KUKA KRL program: MyProgram_001().src

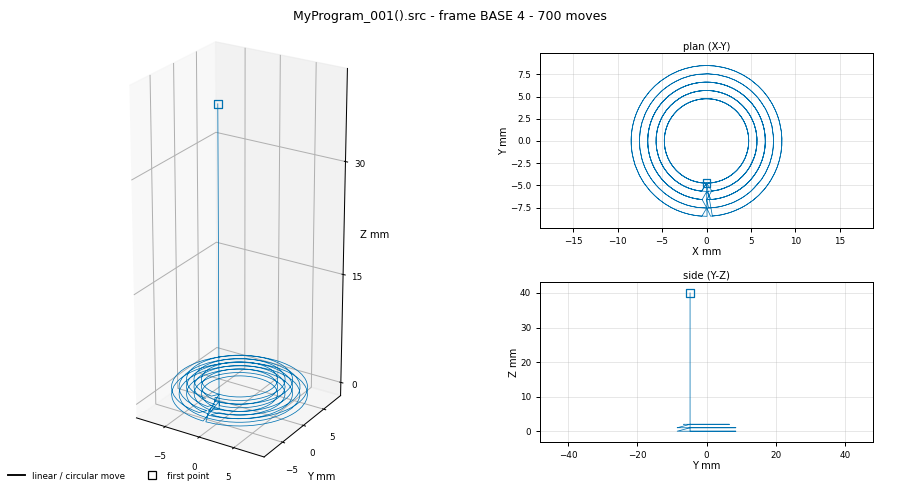
[picture p0: tool path of MyProgram_001().src in frame BASE 4, 700 of 700 moves have a stored position in this frame; points joined in program order, loops and branches not executed]
&ACCESS RVP
&REL 1
&PARAM TEMPLATE = C:\KRC\Roboter\Template\vorgabe
&PARAM EDITMASK = *
DEF MyProgram_001()
; ---- Setting reference (Base) ----
$BASE = BASE_DATA[4]

; --------------------------
; ---- Setting tool (TCP) ----
$TOOL = TOOL_DATA[3]
; --------------------------

$VEL.CP = VEL_APROX_PRINT
LIN {X 0.0001,Y -4.7575,Z 40,A -2.9196,B 0,C 0,E1 0.1598,E2 90.075} C_DIS
LIN {X 0.0001,Y -4.7575,Z 20,A -2.9741,B 0,C 0,E1 0.1598,E2 90.0715} C_DIS
LIN {X 0.0001,Y -4.7574,Z 5,A -3.0236,B 0,C 0,E1 0.1598,E2 90.0708} C_DIS
LIN {X 0.0001,Y -4.7574,Z 0,A -3.042,B 0,C 0,E1 0.1598,E2 90.0712} C_DIS
Startdeposition()
$VEL.CP = VEL_PRINT
LIN {X 0.729,Y -4.6967,Z 0,A -3.013,B 0,C 0,E1 0.1598,E2 90.0715} C_DIS
LIN {X 1.3006,Y -4.5717,Z 0,A -2.9867,B 0,C 0,E1 0.1598,E2 90.0715} C_DIS
LIN {X 1.852,Y -4.3758,Z 0,A -2.9582,B 0,C 0,E1 0.1598,E2 90.0716} C_DIS
LIN {X 2.3763,Y -4.1161,Z 0,A -2.9279,B 0,C 0,E1 0.1598,E2 90.0716} C_DIS
LIN {X 2.863,Y -3.7913,Z 0,A -2.8963,B 0,C 0,E1 0.1598,E2 90.0716} C_DIS
LIN {X 3.3078,Y -3.4112,Z 0,A -2.8639,B 0,C 0,E1 0.1598,E2 90.0716} C_DIS
LIN {X 3.7028,Y -2.9796,Z 0,A -2.8311,B 0,C 0,E1 0.1598,E2 90.0717} C_DIS
LIN {X 4.0408,Y -2.502,Z 0,A -2.7984,B 0,C 0,E1 0.1598,E2 90.0717} C_DIS
LIN {X 4.3736,Y -1.8511,Z 0,A -2.7585,B 0,C 0,E1 0.1598,E2 90.0717} C_DIS
LIN {X 4.6087,Y -1.159,Z 0,A -2.7205,B 0,C 0,E1 0.1598,E2 90.0717} C_DIS
LIN {X 4.7149,Y -0.5836,Z 0,A -2.6923,B 0,C 0,E1 0.1598,E2 90.0718} C_DIS
LIN {X 4.7532,Y 0.0001,Z 0,A -2.6662,B 0,C 0,E1 0.1598,E2 90.0718} C_DIS
LIN {X 4.7174,Y 0.5841,Z 0,A -2.6428,B 0,C 0,E1 0.1598,E2 90.0718} C_DIS
LIN {X 4.6082,Y 1.159,Z 0,A -2.6225,B 0,C 0,E1 0.1598,E2 90.0718} C_DIS
LIN {X 4.432,Y 1.717,Z 0,A -2.6054,B 0,C 0,E1 0.1598,E2 90.0719} C_DIS
LIN {X 4.1869,Y 2.2483,Z 0,A -2.5919,B 0,C 0,E1 0.1598,E2 90.0719} C_DIS
LIN {X 3.8798,Y 2.7464,Z 0,A -2.5822,B 0,C 0,E1 0.1598,E2 90.0719} C_DIS
LIN {X 3.5129,Y 3.2022,Z 0,A -2.5765,B 0,C 0,E1 0.1598,E2 90.072} C_DIS
LIN {X 3.093,Y 3.6098,Z 0,A -2.5748,B 0,C 0,E1 0.1598,E2 90.072} C_DIS
LIN {X 2.6244,Y 3.96,Z 0,A -2.5773,B 0,C 0,E1 0.1598,E2 90.072} C_DIS
LIN {X 2.1186,Y 4.2543,Z 0,A -2.5835,B 0,C 0,E1 0.1598,E2 90.072} C_DIS
LIN {X 1.5797,Y 4.4822,Z 0,A -2.5938,B 0,C 0,E1 0.1598,E2 90.072} C_DIS
LIN {X 1.0171,Y 4.6432,Z 0,A -2.6077,B 0,C 0,E1 0.1598,E2 90.072} C_DIS
LIN {X 0.4388,Y 4.7328,Z 0,A -2.6253,B 0,C 0,E1 0.1598,E2 90.072} C_DIS
LIN {X -0.146,Y 4.7489,Z 0,A -2.6462,B 0,C 0,E1 0.1598,E2 90.072} C_DIS
LIN {X -0.7286,Y 4.6955,Z 0,A -2.6699,B 0,C 0,E1 0.1598,E2 90.072} C_DIS
LIN {X -1.2999,Y 4.5696,Z 0,A -2.6963,B 0,C 0,E1 0.1598,E2 90.072} C_DIS
LIN {X -1.8518,Y 4.3757,Z 0,A -2.7248,B 0,C 0,E1 0.1598,E2 90.072} C_DIS
LIN {X -2.3762,Y 4.1162,Z 0,A -2.7551,B 0,C 0,E1 0.1598,E2 90.0719} C_DIS
LIN {X -2.8631,Y 3.7917,Z 0,A -2.7866,B 0,C 0,E1 0.1598,E2 90.0719} C_DIS
LIN {X -3.3074,Y 3.4109,Z 0,A -2.819,B 0,C 0,E1 0.1598,E2 90.0718} C_DIS
LIN {X -3.7024,Y 2.9793,Z 0,A -2.8517,B 0,C 0,E1 0.1598,E2 90.0717} C_DIS
LIN {X -4.0411,Y 2.5023,Z 0,A -2.8843,B 0,C 0,E1 0.1598,E2 90.0717} C_DIS
LIN {X -4.3161,Y 1.9857,Z 0,A -2.9161,B 0,C 0,E1 0.1598,E2 90.0716} C_DIS
LIN {X -4.5276,Y 1.4403,Z 0,A -2.9468,B 0,C 0,E1 0.1598,E2 90.0715} C_DIS
LIN {X -4.6724,Y 0.8734,Z 0,A -2.976,B 0,C 0,E1 0.1598,E2 90.0715} C_DIS
LIN {X -4.7426,Y 0.2924,Z 0,A -3.003,B 0,C 0,E1 0.1598,E2 90.0715} C_DIS
LIN {X -4.7423,Y -0.2925,Z 0,A -3.0276,B 0,C 0,E1 0.1598,E2 90.0714} C_DIS
LIN {X -4.6721,Y -0.8734,Z 0,A -3.0495,B 0,C 0,E1 0.1598,E2 90.0714} C_DIS
LIN {X -4.528,Y -1.4404,Z 0,A -3.0681,B 0,C 0,E1 0.1598,E2 90.0714} C_DIS
LIN {X -4.3169,Y -1.986,Z 0,A -3.0833,B 0,C 0,E1 0.1598,E2 90.0714} C_DIS
LIN {X -4.0393,Y -2.501,Z 0,A -3.0949,B 0,C 0,E1 0.1598,E2 90.0714} C_DIS
LIN {X -3.7028,Y -2.9797,Z 0,A -3.1027,B 0,C 0,E1 0.1598,E2 90.0714} C_DIS
LIN {X -3.3089,Y -3.4126,Z 0,A -3.1065,B 0,C 0,E1 0.1598,E2 90.0714} C_DIS
LIN {X -2.8642,Y -3.7927,Z 0,A -3.1062,B 0,C 0,E1 0.1598,E2 90.0714} C_DIS
LIN {X -2.2471,Y -4.1846,Z 0,A -3.1,B 0,C 0,E1 0.1598,E2 90.0714} C_DIS
LIN {X -1.5793,Y -4.482,Z 0,A -3.0881,B 0,C 0,E1 0.1598,E2 90.0714} C_DIS
LIN {X -0.7289,Y -4.6968,Z 0,A -3.066,B 0,C 0,E1 0.1598,E2 90.0714} C_DIS
LIN {X 0.0001,Y -4.7573,Z 0,A -3.0418,B 0,C 0,E1 0.1598,E2 90.0715} C_DIS
Enddeposition()
LIN {X 0.0001,Y -4.7573,Z 0,A -3.0418,B 0,C 0,E1 0.1598,E2 90.0715} C_DIS
Startdeposition()
$VEL.CP = VEL_PRINT
LIN {X -0.5659,Y -5.6552,Z 0,A -3.1001,B 0,C 0,E1 0.1598,E2 90.0709} C_DIS
LIN {X -1.328,Y -5.5261,Z 0,A -3.1231,B 0,C 0,E1 0.1598,E2 90.0714} C_DIS
LIN {X -2.0655,Y -5.2941,Z 0,A -3.1404,B 0,C 0,E1 0.1598,E2 90.0714} C_DIS
LIN {X -2.7651,Y -4.9655,Z 0,A -3.1522,B 0,C 0,E1 0.1598,E2 90.0714} C_DIS
LIN {X -3.4132,Y -4.5441,Z 0,A -3.1582,B 0,C 0,E1 0.1598,E2 90.0713} C_DIS
LIN {X -4.2289,Y -3.8084,Z 0,A -3.1569,B 0,C 0,E1 0.1598,E2 90.0711} C_DIS
LIN {X -4.8665,Y -2.9396,Z 0,A -3.1436,B 0,C 0,E1 0.1598,E2 90.071} C_DIS
LIN {X -5.2026,Y -2.2902,Z 0,A -3.1288,B 0,C 0,E1 0.1598,E2 90.0712} C_DIS
LIN {X -5.4555,Y -1.6043,Z 0,A -3.1092,B 0,C 0,E1 0.1598,E2 90.0712} C_DIS
LIN {X -5.6146,Y -0.8906,Z 0,A -3.085,B 0,C 0,E1 0.1598,E2 90.0712} C_DIS
LIN {X -5.6818,Y -0.1626,Z 0,A -3.0568,B 0,C 0,E1 0.1598,E2 90.0712} C_DIS
LIN {X -5.6568,Y 0.5679,Z 0,A -3.0251,B 0,C 0,E1 0.1598,E2 90.0712} C_DIS
LIN {X -5.5358,Y 1.2889,Z 0,A -2.9904,B 0,C 0,E1 0.1598,E2 90.0713} C_DIS
LIN {X -5.3256,Y 1.989,Z 0,A -2.9532,B 0,C 0,E1 0.1598,E2 90.0713} C_DIS
LIN {X -5.0257,Y 2.6559,Z 0,A -2.9141,B 0,C 0,E1 0.1598,E2 90.0715} C_DIS
LIN {X -4.6436,Y 3.2789,Z 0,A -2.8738,B 0,C 0,E1 0.1598,E2 90.0715} C_DIS
LIN {X -4.183,Y 3.8466,Z 0,A -2.833,B 0,C 0,E1 0.1598,E2 90.0716} C_DIS
LIN {X -3.6562,Y 4.3534,Z 0,A -2.7923,B 0,C 0,E1 0.1598,E2 90.0717} C_DIS
LIN {X -2.6911,Y 5.0128,Z 0,A -2.7289,B 0,C 0,E1 0.1598,E2 90.0717} C_DIS
LIN {X -1.7583,Y 5.405,Z 0,A -2.6781,B 0,C 0,E1 0.1598,E2 90.0719} C_DIS
LIN {X -0.9727,Y 5.6007,Z 0,A -2.6409,B 0,C 0,E1 0.1598,E2 90.072} C_DIS
LIN {X -0.1673,Y 5.6823,Z 0,A -2.6078,B 0,C 0,E1 0.1598,E2 90.072} C_DIS
LIN {X 0.6415,Y 5.6477,Z 0,A -2.5794,B 0,C 0,E1 0.1598,E2 90.0721} C_DIS
LIN {X 1.4369,Y 5.4977,Z 0,A -2.5564,B 0,C 0,E1 0.1598,E2 90.0721} C_DIS
LIN {X 2.2035,Y 5.2384,Z 0,A -2.539,B 0,C 0,E1 0.1598,E2 90.0721} C_DIS
LIN {X 2.9262,Y 4.8736,Z 0,A -2.5277,B 0,C 0,E1 0.1598,E2 90.0721} C_DIS
LIN {X 3.5891,Y 4.409,Z 0,A -2.5228,B 0,C 0,E1 0.1598,E2 90.0721} C_DIS
LIN {X 4.1789,Y 3.8541,Z 0,A -2.5245,B 0,C 0,E1 0.1598,E2 90.0721} C_DIS
LIN {X 4.6838,Y 3.2212,Z 0,A -2.5326,B 0,C 0,E1 0.1598,E2 90.072} C_DIS
LIN {X 5.0948,Y 2.5236,Z 0,A -2.5469,B 0,C 0,E1 0.1598,E2 90.0719} C_DIS
LIN {X 5.4021,Y 1.7745,Z 0,A -2.5673,B 0,C 0,E1 0.1598,E2 90.0719} C_DIS
LIN {X 5.5992,Y 0.9892,Z 0,A -2.5932,B 0,C 0,E1 0.1598,E2 90.0718} C_DIS
LIN {X 5.6822,Y 0.1837,Z 0,A -2.6242,B 0,C 0,E1 0.1598,E2 90.0718} C_DIS
LIN {X 5.6508,Y -0.6252,Z 0,A -2.6597,B 0,C 0,E1 0.1598,E2 90.0717} C_DIS
LIN {X 5.4551,Y -1.6182,Z 0,A -2.7087,B 0,C 0,E1 0.1598,E2 90.0714} C_DIS
LIN {X 4.7566,Y -3.1241,Z 0,A -2.7976,B 0,C 0,E1 0.1598,E2 90.0708} C_DIS
LIN {X 4.1077,Y -3.9363,Z 0,A -2.8565,B 0,C 0,E1 0.1598,E2 90.0714} C_DIS
LIN {X 3.4756,Y -4.4996,Z 0,A -2.9038,B 0,C 0,E1 0.1598,E2 90.0716} C_DIS
LIN {X 2.6266,Y -5.0483,Z 0,A -2.9583,B 0,C 0,E1 0.1598,E2 90.0715} C_DIS
LIN {X 1.4839,Y -5.4928,Z 0,A -3.0191,B 0,C 0,E1 0.1598,E2 90.0715} C_DIS
LIN {X 0.5699,Y -5.656,Z 0,A -3.0596,B 0,C 0,E1 0.1598,E2 90.0715} C_DIS
LIN {X 0.5699,Y -5.656,Z 0,A -3.0596,B 0,C 0,E1 0.1598,E2 90.0715} C_DIS
Enddeposition()
LIN {X 0.0153,Y -6.6202,Z 0,A -3.1197,B 0,C 0,E1 0.1598,E2 90.0703} C_DIS
Startdeposition()
$VEL.CP = VEL_PRINT
LIN {X 0.8653,Y -6.5643,Z 0,A -3.0873,B 0,C 0,E1 0.1598,E2 90.0714} C_DIS
LIN {X 1.5356,Y -6.4404,Z 0,A -3.0575,B 0,C 0,E1 0.1598,E2 90.0714} C_DIS
LIN {X 2.1897,Y -6.2485,Z 0,A -3.0253,B 0,C 0,E1 0.1598,E2 90.0715} C_DIS
LIN {X 2.8206,Y -5.9905,Z 0,A -2.9913,B 0,C 0,E1 0.1598,E2 90.0715} C_DIS
LIN {X 3.4216,Y -5.6688,Z 0,A -2.9556,B 0,C 0,E1 0.1598,E2 90.0715} C_DIS
LIN {X 3.9851,Y -5.2852,Z 0,A -2.9186,B 0,C 0,E1 0.1598,E2 90.0716} C_DIS
LIN {X 4.5088,Y -4.849,Z 0,A -2.8809,B 0,C 0,E1 0.1598,E2 90.0716} C_DIS
LIN {X 4.9834,Y -4.3597,Z 0,A -2.8427,B 0,C 0,E1 0.1598,E2 90.0716} C_DIS
LIN {X 5.4053,Y -3.8243,Z 0,A -2.8045,B 0,C 0,E1 0.1598,E2 90.0716} C_DIS
LIN {X 5.7689,Y -3.2476,Z 0,A -2.7666,B 0,C 0,E1 0.1598,E2 90.0717} C_DIS
LIN {X 6.0736,Y -2.6379,Z 0,A -2.7296,B 0,C 0,E1 0.1598,E2 90.0717} C_DIS
LIN {X 6.3126,Y -1.9995,Z 0,A -2.6937,B 0,C 0,E1 0.1598,E2 90.0717} C_DIS
LIN {X 6.4835,Y -1.3396,Z 0,A -2.6594,B 0,C 0,E1 0.1598,E2 90.0717} C_DIS
LIN {X 6.586,Y -0.6656,Z 0,A -2.6271,B 0,C 0,E1 0.1598,E2 90.0718} C_DIS
LIN {X 6.6196,Y 0.0151,Z 0,A -2.597,B 0,C 0,E1 0.1598,E2 90.0718} C_DIS
LIN {X 6.5847,Y 0.6959,Z 0,A -2.5694,B 0,C 0,E1 0.1598,E2 90.0718} C_DIS
LIN {X 6.4794,Y 1.3694,Z 0,A -2.5448,B 0,C 0,E1 0.1598,E2 90.0719} C_DIS
LIN {X 6.3031,Y 2.0279,Z 0,A -2.5234,B 0,C 0,E1 0.1598,E2 90.0719} C_DIS
LIN {X 6.0589,Y 2.6644,Z 0,A -2.5055,B 0,C 0,E1 0.1598,E2 90.072} C_DIS
LIN {X 5.7524,Y 3.2732,Z 0,A -2.491,B 0,C 0,E1 0.1598,E2 90.072} C_DIS
LIN {X 5.3874,Y 3.8487,Z 0,A -2.4801,B 0,C 0,E1 0.1598,E2 90.072} C_DIS
LIN {X 4.9631,Y 4.3822,Z 0,A -2.4732,B 0,C 0,E1 0.1598,E2 90.0721} C_DIS
LIN {X 4.486,Y 4.8689,Z 0,A -2.4703,B 0,C 0,E1 0.1598,E2 90.0721} C_DIS
LIN {X 3.9617,Y 5.3048,Z 0,A -2.4712,B 0,C 0,E1 0.1598,E2 90.0721} C_DIS
LIN {X 3.3953,Y 5.6842,Z 0,A -2.4761,B 0,C 0,E1 0.1598,E2 90.0721} C_DIS
LIN {X 2.7929,Y 6.0031,Z 0,A -2.4849,B 0,C 0,E1 0.1598,E2 90.0721} C_DIS
LIN {X 2.1607,Y 6.2576,Z 0,A -2.4975,B 0,C 0,E1 0.1598,E2 90.0721} C_DIS
LIN {X 1.5056,Y 6.4462,Z 0,A -2.5137,B 0,C 0,E1 0.1598,E2 90.0721} C_DIS
LIN {X 0.8347,Y 6.5669,Z 0,A -2.5334,B 0,C 0,E1 0.1598,E2 90.0721} C_DIS
LIN {X 0.1551,Y 6.6205,Z 0,A -2.5563,B 0,C 0,E1 0.1598,E2 90.0721} C_DIS
LIN {X -0.5262,Y 6.5998,Z 0,A -2.5823,B 0,C 0,E1 0.1598,E2 90.0721} C_DIS
LIN {X -1.202,Y 6.51,Z 0,A -2.611,B 0,C 0,E1 0.1598,E2 90.0721} C_DIS
LIN {X -1.865,Y 6.3515,Z 0,A -2.6421,B 0,C 0,E1 0.1598,E2 90.0721} C_DIS
LIN {X -2.5085,Y 6.1267,Z 0,A -2.6753,B 0,C 0,E1 0.1598,E2 90.072} C_DIS
LIN {X -3.1256,Y 5.8372,Z 0,A -2.7103,B 0,C 0,E1 0.1598,E2 90.072} C_DIS
LIN {X -3.7086,Y 5.4841,Z 0,A -2.7466,B 0,C 0,E1 0.1598,E2 90.0719} C_DIS
LIN {X -4.2535,Y 5.0745,Z 0,A -2.7839,B 0,C 0,E1 0.1598,E2 90.0718} C_DIS
LIN {X -4.7527,Y 4.6103,Z 0,A -2.8218,B 0,C 0,E1 0.1598,E2 90.0718} C_DIS
LIN {X -5.2014,Y 4.0972,Z 0,A -2.8599,B 0,C 0,E1 0.1598,E2 90.0716} C_DIS
LIN {X -5.5952,Y 3.5407,Z 0,A -2.8978,B 0,C 0,E1 0.1598,E2 90.0716} C_DIS
LIN {X -5.9297,Y 2.9468,Z 0,A -2.9351,B 0,C 0,E1 0.1598,E2 90.0715} C_DIS
LIN {X -6.1988,Y 2.3205,Z 0,A -2.9713,B 0,C 0,E1 0.1598,E2 90.0715} C_DIS
LIN {X -6.4043,Y 1.6707,Z 0,A -3.0061,B 0,C 0,E1 0.1598,E2 90.0714} C_DIS
LIN {X -6.5434,Y 1.0033,Z 0,A -3.0393,B 0,C 0,E1 0.1598,E2 90.0713} C_DIS
LIN {X -6.6132,Y 0.3254,Z 0,A -3.0704,B 0,C 0,E1 0.1598,E2 90.0713} C_DIS
LIN {X -6.6118,Y -0.3563,Z 0,A -3.099,B 0,C 0,E1 0.1598,E2 90.0713} C_DIS
LIN {X -6.5412,Y -1.0343,Z 0,A -3.1249,B 0,C 0,E1 0.1598,E2 90.0712} C_DIS
LIN {X -6.3998,Y -1.7012,Z 0,A -3.1478,B 0,C 0,E1 0.1598,E2 90.0712} C_DIS
LIN {X -6.1902,Y -2.3499,Z 0,A -3.1674,B 0,C 0,E1 0.1598,E2 90.0712} C_DIS
LIN {X -5.9153,Y -2.9737,Z 0,A -3.1835,B 0,C 0,E1 0.1598,E2 90.0712} C_DIS
LIN {X -5.5783,Y -3.5663,Z 0,A -3.1961,B 0,C 0,E1 0.1598,E2 90.0712} C_DIS
LIN {X -5.1816,Y -4.1206,Z 0,A -3.2049,B 0,C 0,E1 0.1598,E2 90.0712} C_DIS
LIN {X -4.7309,Y -4.632,Z 0,A -3.21,B 0,C 0,E1 0.1598,E2 90.0712} C_DIS
LIN {X -4.2296,Y -5.0939,Z 0,A -3.211,B 0,C 0,E1 0.1598,E2 90.0712} C_DIS
LIN {X -3.6835,Y -5.5018,Z 0,A -3.2082,B 0,C 0,E1 0.1598,E2 90.0712} C_DIS
LIN {X -3.0976,Y -5.8502,Z 0,A -3.2014,B 0,C 0,E1 0.1598,E2 90.0712} C_DIS
LIN {X -2.4799,Y -6.1385,Z 0,A -3.191,B 0,C 0,E1 0.1598,E2 90.0712} C_DIS
LIN {X -1.8357,Y -6.3613,Z 0,A -3.1768,B 0,C 0,E1 0.1598,E2 90.0713} C_DIS
LIN {X -1.172,Y -6.5165,Z 0,A -3.159,B 0,C 0,E1 0.1598,E2 90.0713} C_DIS
LIN {X -0.4958,Y -6.6018,Z 0,A -3.1378,B 0,C 0,E1 0.1598,E2 90.0713} C_DIS
LIN {X -0.4958,Y -6.6018,Z 0,A -3.1378,B 0,C 0,E1 0.1598,E2 90.0713} C_DIS
Enddeposition()
LIN {X 0.0326,Y -7.5539,Z 0,A -3.5262,B 0,C 0.001,E1 0.1598,E2 90.4405} C_DIS
Startdeposition()
$VEL.CP = VEL_PRINT
LIN {X -1.0951,Y -7.4778,Z 0,A -3.5603,B -0.0001,C 0.001,E1 0.1596,E2 90.4361} C_DIS
LIN {X -2.1091,Y -7.2579,Z 0,A -3.5757,B -0.0003,C 0.001,E1 0.1595,E2 90.4233} C_DIS
LIN {X -3.0894,Y -6.8977,Z 0,A -3.5778,B -0.0003,C 0.001,E1 0.1593,E2 90.4042} C_DIS
LIN {X -3.9943,Y -6.4145,Z 0,A -3.5667,B -0.0005,C 0.0009,E1 0.1593,E2 90.38} C_DIS
LIN {X -4.8258,Y -5.8109,Z 0,A -3.5431,B -0.0006,C 0.0009,E1 0.1591,E2 90.351} C_DIS
LIN {X -5.6854,Y -4.9782,Z 0,A -3.4974,B -0.0008,C 0.0007,E1 0.159,E2 90.3086} C_DIS
LIN {X -6.225,Y -4.2757,Z 0,A -3.4544,B -0.0008,C 0.0007,E1 0.159,E2 90.2753} C_DIS
LIN {X -6.5998,Y -3.6743,Z 0,A -3.4129,B -0.0008,C 0.0005,E1 0.1589,E2 90.2453} C_DIS
LIN {X -6.916,Y -3.0399,Z 0,A -3.3655,B -0.0009,C 0.0005,E1 0.1589,E2 90.213} C_DIS
LIN {X -7.2264,Y -2.2101,Z 0,A -3.2968,B -0.0009,C 0.0003,E1 0.1588,E2 90.1679} C_DIS
LIN {X -7.4885,Y -0.9844,Z 0,A -3.1954,B -0.001,C 0.0002,E1 0.1588,E2 90.1086} C_DIS
LIN {X -7.5539,Y 0.2224,Z 0,A -3.0846,B -0.001,C 0,E1 0.1588,E2 90.0466} C_DIS
LIN {X -7.4567,Y 1.2263,Z 0,A -2.9913,B -0.001,C -0.0001,E1 0.1588,E2 89.9994} C_DIS
LIN {X -7.2768,Y 2.0424,Z 0,A -2.9087,B -0.001,C -0.0003,E1 0.1588,E2 89.9581} C_DIS
LIN {X -6.9542,Y 2.9565,Z 0,A -2.8142,B -0.001,C -0.0003,E1 0.1588,E2 89.9143} C_DIS
LIN {X -6.3784,Y 4.0527,Z 0,A -2.6949,B -0.0009,C -0.0005,E1 0.1589,E2 89.8628} C_DIS
LIN {X -5.7875,Y 4.8589,Z 0,A -2.5995,B -0.0008,C -0.0007,E1 0.159,E2 89.8234} C_DIS
LIN {X -4.9697,Y 5.6869,Z 0,A -2.497,B -0.0007,C -0.0007,E1 0.1591,E2 89.7862} C_DIS
LIN {X -3.9421,Y 6.4467,Z 0,A -2.3915,B -0.0006,C -0.0009,E1 0.1593,E2 89.7509} C_DIS
LIN {X -2.8085,Y 7.0171,Z 0,A -2.2981,B -0.0004,C -0.0009,E1 0.1594,E2 89.7233} C_DIS
LIN {X -1.8335,Y 7.3312,Z 0,A -2.2359,B -0.0003,C -0.001,E1 0.1596,E2 89.7103} C_DIS
LIN {X -0.9234,Y 7.5006,Z 0,A -2.1887,B -0.0001,C -0.001,E1 0.1597,E2 89.7037} C_DIS
LIN {X 0.2516,Y 7.5494,Z 0,A -2.1431,B 0,C -0.001,E1 0.1599,E2 89.7033} C_DIS
LIN {X 1.2917,Y 7.4461,Z 0,A -2.1167,B 0.0002,C -0.001,E1 0.16,E2 89.7106} C_DIS
LIN {X 2.3706,Y 7.1703,Z 0,A -2.1034,B 0.0003,C -0.001,E1 0.1601,E2 89.7252} C_DIS
LIN {X 3.1224,Y 6.8765,Z 0,A -2.1032,B 0.0004,C -0.001,E1 0.1602,E2 89.74} C_DIS
LIN {X 3.8388,Y 6.5046,Z 0,A -2.1124,B 0.0005,C -0.0009,E1 0.1603,E2 89.7597} C_DIS
LIN {X 4.5113,Y 6.0581,Z 0,A -2.1294,B 0.0006,C -0.0009,E1 0.1604,E2 89.7824} C_DIS
LIN {X 5.1327,Y 5.5427,Z 0,A -2.155,B 0.0006,C -0.0008,E1 0.1605,E2 89.8089} C_DIS
LIN {X 5.8282,Y 4.8113,Z 0,A -2.2023,B 0.0008,C -0.0007,E1 0.1606,E2 89.8507} C_DIS
LIN {X 6.599,Y 3.6818,Z 0,A -2.2727,B 0.0008,C -0.0005,E1 0.1607,E2 89.9015} C_DIS
LIN {X 7.0112,Y 2.8219,Z 0,A -2.342,B 0.001,C -0.0004,E1 0.1607,E2 89.9496} C_DIS
LIN {X 7.374,Y 1.6552,Z 0,A -2.428,B 0.001,C -0.0002,E1 0.1608,E2 89.9996} C_DIS
LIN {X 7.5565,Y 0.107,Z 0,A -2.5763,B 0.001,C 0,E1 0.1608,E2 90.0893} C_DIS
LIN {X 7.4445,Y -1.3018,Z 0,A -2.7007,B 0.001,C 0.0002,E1 0.1608,E2 90.1502} C_DIS
LIN {X 7.1255,Y -2.5177,Z 0,A -2.8212,B 0.001,C 0.0003,E1 0.1608,E2 90.2078} C_DIS
LIN {X 6.6617,Y -3.5611,Z 0,A -2.9251,B 0.001,C 0.0005,E1 0.1607,E2 90.2507} C_DIS
LIN {X 6.2296,Y -4.2769,Z 0,A -3.0183,B 0.0008,C 0.0005,E1 0.1607,E2 90.298} C_DIS
LIN {X 4.991,Y -5.6745,Z 0,A -3.1799,B 0.0007,C 0.0008,E1 0.1605,E2 90.3552} C_DIS
LIN {X 4.2679,Y -6.2306,Z 0,A -3.2545,B 0.0007,C 0.0008,E1 0.1604,E2 90.3798} C_DIS
LIN {X 3.6468,Y -6.6137,Z 0,A -3.312,B 0.0005,C 0.0008,E1 0.1603,E2 90.3983} C_DIS
LIN {X 2.825,Y -7.0101,Z 0,A -3.38,B 0.0004,C 0.001,E1 0.1601,E2 90.4193} C_DIS
LIN {X 1.677,Y -7.3653,Z 0,A -3.4513,B 0.0003,C 0.001,E1 0.16,E2 90.4333} C_DIS
LIN {X 0.9514,Y -7.4929,Z 0,A -3.489,B 0.0002,C 0.001,E1 0.1599,E2 90.4388} C_DIS
LIN {X 0.0326,Y -7.5539,Z 0,A -3.5277,B 0.0001,C 0.001,E1 0.1599,E2 90.441} C_DIS
Enddeposition()
LIN {X 0.0326,Y -7.5539,Z 0,A -3.5277,B 0.0001,C 0.001,E1 0.1599,E2 90.441} C_DIS
Startdeposition()
$VEL.CP = VEL_PRINT
LIN {X 0.4573,Y -8.4789,Z 0,A -3.5765,B 0.0001,C 0.001,E1 0.1599,E2 90.4664} C_DIS
LIN {X 1.6933,Y -8.3185,Z 0,A -3.5159,B 0.0003,C 0.001,E1 0.16,E2 90.4582} C_DIS
LIN {X 2.6816,Y -8.0571,Z 0,A -3.4528,B 0.0005,C 0.001,E1 0.1602,E2 90.4426} C_DIS
LIN {X 3.8165,Y -7.5813,Z 0,A -3.3691,B 0.0005,C 0.001,E1 0.1603,E2 90.4208} C_DIS
LIN {X 4.5456,Y -7.1686,Z 0,A -3.3045,B 0.0007,C 0.0009,E1 0.1604,E2 90.4004} C_DIS
LIN {X 5.2304,Y -6.6859,Z 0,A -3.2355,B 0.0007,C 0.0009,E1 0.1604,E2 90.3769} C_DIS
LIN {X 5.8643,Y -6.1381,Z 0,A -3.1628,B 0.0008,C 0.0007,E1 0.1606,E2 90.3506} C_DIS
LIN {X 6.6486,Y -5.2813,Z 0,A -3.0546,B 0.0009,C 0.0007,E1 0.1606,E2 90.3072} C_DIS
LIN {X 7.2756,Y -4.3694,Z 0,A -2.9512,B 0.0009,C 0.0005,E1 0.1608,E2 90.2653} C_DIS
LIN {X 7.6576,Y -3.6565,Z 0,A -2.8749,B 0.001,C 0.0005,E1 0.1608,E2 90.2329} C_DIS
LIN {X 7.971,Y -2.911,Z 0,A -2.7969,B 0.001,C 0.0003,E1 0.1608,E2 90.1978} C_DIS
LIN {X 8.2122,Y -2.139,Z 0,A -2.7194,B 0.001,C 0.0003,E1 0.1608,E2 90.1617} C_DIS
LIN {X 8.379,Y -1.3476,Z 0,A -2.6431,B 0.0011,C 0.0001,E1 0.1608,E2 90.1249} C_DIS
LIN {X 8.4699,Y -0.5439,Z 0,A -2.5686,B 0.0011,C 0,E1 0.1609,E2 90.0876} C_DIS
LIN {X 8.4843,Y 0.2648,Z 0,A -2.4957,B 0.0011,C -0.0001,E1 0.1609,E2 90.0493} C_DIS
LIN {X 8.4203,Y 1.0712,Z 0,A -2.4268,B 0.0011,C -0.0002,E1 0.1609,E2 90.0121} C_DIS
LIN {X 8.1807,Y 2.2762,Z 0,A -2.3283,B 0.0011,C -0.0004,E1 0.1609,E2 89.9558} C_DIS
LIN {X 7.8752,Y 3.1763,Z 0,A -2.2576,B 0.001,C -0.0004,E1 0.1609,E2 89.912} C_DIS
LIN {X 7.4082,Y 4.1479,Z 0,A -2.1908,B 0.001,C -0.0006,E1 0.1607,E2 89.8691} C_DIS
LIN {X 6.8716,Y 4.9798,Z 0,A -2.1378,B 0.0009,C -0.0007,E1 0.1607,E2 89.8317} C_DIS
LIN {X 6.3781,Y 5.5993,Z 0,A -2.1029,B 0.0008,C -0.0007,E1 0.1607,E2 89.805} C_DIS
LIN {X 5.8299,Y 6.1708,Z 0,A -2.0717,B 0.0008,C -0.0009,E1 0.1605,E2 89.778} C_DIS
LIN {X 4.9715,Y 6.8844,Z 0,A -2.0396,B 0.0006,C -0.0009,E1 0.1605,E2 89.7447} C_DIS
LIN {X 3.9276,Y 7.5292,Z 0,A -2.0205,B 0.0004,C -0.001,E1 0.1603,E2 89.7148} C_DIS
LIN {X 3.0806,Y 7.9132,Z 0,A -2.0179,B 0.0004,C -0.001,E1 0.1602,E2 89.6975} C_DIS
LIN {X 2.0657,Y 8.2355,Z 0,A -2.0277,B 0.0002,C -0.001,E1 0.16,E2 89.6838} C_DIS
LIN {X 0.8504,Y 8.4438,Z 0,A -2.0556,B 0,C -0.0011,E1 0.1599,E2 89.676} C_DIS
LIN {X 0.0341,Y 8.4871,Z 0,A -2.0824,B 0,C -0.0011,E1 0.1598,E2 89.6747} C_DIS
LIN {X -0.7826,Y 8.4504,Z 0,A -2.1163,B -0.0002,C -0.0011,E1 0.1597,E2 89.6771} C_DIS
LIN {X -1.592,Y 8.3354,Z 0,A -2.1569,B -0.0002,C -0.0011,E1 0.1596,E2 89.6831} C_DIS
LIN {X -2.3866,Y 8.1432,Z 0,A -2.2038,B -0.0004,C -0.0011,E1 0.1595,E2 89.6927} C_DIS
LIN {X -3.1595,Y 7.8764,Z 0,A -2.2567,B -0.0004,C -0.0011,E1 0.1594,E2 89.7058} C_DIS
LIN {X -4.085,Y 7.4427,Z 0,A -2.3317,B -0.0006,C -0.0009,E1 0.1592,E2 89.7283} C_DIS
LIN {X -5.1035,Y 6.7819,Z 0,A -2.4216,B -0.0007,C -0.0009,E1 0.1592,E2 89.7527} C_DIS
LIN {X -5.7314,Y 6.2655,Z 0,A -2.4968,B -0.0008,C -0.0008,E1 0.159,E2 89.7828} C_DIS
LIN {X -6.3932,Y 5.587,Z 0,A -2.5851,B -0.0008,C -0.0007,E1 0.159,E2 89.8178} C_DIS
LIN {X -7.0154,Y 4.7753,Z 0,A -2.6796,B -0.001,C -0.0006,E1 0.1589,E2 89.8549} C_DIS
LIN {X -7.4425,Y 4.0776,Z 0,A -2.7584,B -0.001,C -0.0005,E1 0.1589,E2 89.8883} C_DIS
LIN {X -7.8005,Y 3.3419,Z 0,A -2.8377,B -0.001,C -0.0004,E1 0.1588,E2 89.9232} C_DIS
LIN {X -8.0862,Y 2.5753,Z 0,A -2.9171,B -0.001,C -0.0003,E1 0.1588,E2 89.9595} C_DIS
LIN {X -8.297,Y 1.7848,Z 0,A -2.9957,B -0.0011,C -0.0002,E1 0.1587,E2 89.9968} C_DIS
LIN {X -8.431,Y 0.9777,Z 0,A -3.0728,B -0.0011,C 0,E1 0.1587,E2 90.0347} C_DIS
LIN {X -8.487,Y 0.1614,Z 0,A -3.1484,B -0.0011,C 0,E1 0.1587,E2 90.0736} C_DIS
LIN {X -8.4629,Y -0.6565,Z 0,A -3.2209,B -0.0011,C 0.0002,E1 0.1587,E2 90.1124} C_DIS
LIN {X -8.3602,Y -1.4682,Z 0,A -3.2894,B -0.0011,C 0.0002,E1 0.1587,E2 90.1503} C_DIS
LIN {X -8.0608,Y -2.6697,Z 0,A -3.3901,B -0.0011,C 0.0004,E1 0.1587,E2 90.2114} C_DIS
LIN {X -7.5809,Y -3.818,Z 0,A -3.4691,B -0.0009,C 0.0006,E1 0.1588,E2 90.2596} C_DIS
LIN {X -7.0606,Y -4.7166,Z 0,A -3.5318,B -0.0009,C 0.0006,E1 0.1588,E2 90.3036} C_DIS
LIN {X -6.3897,Y -5.5832,Z 0,A -3.5814,B -0.0008,C 0.0008,E1 0.159,E2 90.3416} C_DIS
LIN {X -5.8439,Y -6.1523,Z 0,A -3.6109,B -0.0007,C 0.0008,E1 0.159,E2 90.3673} C_DIS
LIN {X -5.2476,Y -6.6681,Z 0,A -3.634,B -0.0007,C 0.0009,E1 0.1591,E2 90.3908} C_DIS
LIN {X -4.6065,Y -7.1271,Z 0,A -3.6496,B -0.0005,C 0.0009,E1 0.1592,E2 90.4108} C_DIS
LIN {X -3.9256,Y -7.5245,Z 0,A -3.6599,B -0.0005,C 0.001,E1 0.1593,E2 90.4296} C_DIS
LIN {X -3.21,Y -7.8555,Z 0,A -3.6615,B -0.0003,C 0.001,E1 0.1593,E2 90.4437} C_DIS
LIN {X -2.4671,Y -8.1197,Z 0,A -3.6564,B -0.0003,C 0.001,E1 0.1595,E2 90.455} C_DIS
LIN {X -1.7031,Y -8.3142,Z 0,A -3.6443,B -0.0001,C 0.0011,E1 0.1595,E2 90.463} C_DIS
LIN {X -0.9243,Y -8.4373,Z 0,A -3.6253,B -0.0001,C 0.0011,E1 0.1597,E2 90.4677} C_DIS
LIN {X 0.0598,Y -8.4905,Z 0,A -3.5924,B 0.0001,C 0.0011,E1 0.1597,E2 90.4689} C_DIS
Enddeposition()
LIN {X 0.0001,Y -4.7537,Z 1,A -3.0256,B 0.0001,C 0,E1 0.1598,E2 90.0603} C_DIS
Startdeposition()
$VEL.CP = VEL_PRINT
LIN {X 0.0001,Y -4.7537,Z 1,A -3.0313,B 0.0001,C 0,E1 0.1598,E2 90.066} C_DIS
LIN {X -0.6585,Y -4.7075,Z 1,A -3.0583,B 0.0001,C 0,E1 0.1598,E2 90.0708} C_DIS
LIN {X -1.1767,Y -4.6049,Z 1,A -3.0736,B 0.0001,C 0,E1 0.1598,E2 90.0714} C_DIS
LIN {X -1.6807,Y -4.4465,Z 1,A -3.0855,B 0,C 0,E1 0.1598,E2 90.0714} C_DIS
LIN {X -2.1636,Y -4.2321,Z 1,A -3.0941,B 0,C 0,E1 0.1598,E2 90.0714} C_DIS
LIN {X -2.6192,Y -3.9644,Z 1,A -3.0996,B 0,C 0,E1 0.1598,E2 90.0714} C_DIS
LIN {X -3.0442,Y -3.6508,Z 1,A -3.1019,B 0,C 0,E1 0.1598,E2 90.0714} C_DIS
LIN {X -3.4314,Y -3.2914,Z 1,A -3.101,B 0,C 0,E1 0.1598,E2 90.0714} C_DIS
LIN {X -3.7746,Y -2.8897,Z 1,A -3.0966,B 0,C 0,E1 0.1598,E2 90.0714} C_DIS
LIN {X -4.0712,Y -2.4525,Z 1,A -3.0891,B 0,C 0,E1 0.1598,E2 90.0714} C_DIS
LIN {X -4.3172,Y -1.985,Z 1,A -3.0784,B 0,C 0,E1 0.1598,E2 90.0714} C_DIS
LIN {X -4.5121,Y -1.494,Z 1,A -3.0649,B 0,C 0,E1 0.1598,E2 90.0714} C_DIS
LIN {X -4.6488,Y -0.9837,Z 1,A -3.0484,B 0,C 0,E1 0.1598,E2 90.0714} C_DIS
LIN {X -4.7294,Y -0.4618,Z 1,A -3.0294,B 0,C 0,E1 0.1598,E2 90.0714} C_DIS
LIN {X -4.753,Y 0.066,Z 1,A -3.008,B 0,C 0,E1 0.1598,E2 90.0714} C_DIS
LIN {X -4.7169,Y 0.5931,Z 1,A -2.9845,B 0,C 0,E1 0.1598,E2 90.0714} C_DIS
LIN {X -4.621,Y 1.1127,Z 1,A -2.9591,B 0,C 0,E1 0.1598,E2 90.0714} C_DIS
LIN {X -4.4686,Y 1.6186,Z 1,A -2.9322,B 0,C 0,E1 0.1598,E2 90.0715} C_DIS
LIN {X -4.2619,Y 2.1048,Z 1,A -2.9041,B 0,C 0,E1 0.1598,E2 90.0715} C_DIS
LIN {X -4.0025,Y 2.5651,Z 1,A -2.8752,B 0,C 0,E1 0.1598,E2 90.0716} C_DIS
LIN {X -3.6928,Y 2.993,Z 1,A -2.8458,B 0,C 0,E1 0.1598,E2 90.0716} C_DIS
LIN {X -3.3382,Y 3.3846,Z 1,A -2.8162,B 0,C 0,E1 0.1598,E2 90.0717} C_DIS
LIN {X -2.9422,Y 3.7344,Z 1,A -2.7869,B 0,C 0,E1 0.1598,E2 90.0717} C_DIS
LIN {X -2.5082,Y 4.0356,Z 1,A -2.7583,B 0,C 0,E1 0.1598,E2 90.0719} C_DIS
LIN {X -2.0449,Y 4.2893,Z 1,A -2.7305,B 0,C 0,E1 0.1598,E2 90.0719} C_DIS
LIN {X -1.5564,Y 4.4904,Z 1,A -2.704,B 0,C 0,E1 0.1598,E2 90.0719} C_DIS
LIN {X -1.0481,Y 4.6341,Z 1,A -2.6793,B 0,C 0,E1 0.1598,E2 90.0719} C_DIS
LIN {X -0.5275,Y 4.7229,Z 1,A -2.6563,B 0,C 0,E1 0.1598,E2 90.072} C_DIS
LIN {X -0.0001,Y 4.7538,Z 1,A -2.6356,B 0,C 0,E1 0.1598,E2 90.072} C_DIS
LIN {X 0.5273,Y 4.7241,Z 1,A -2.6174,B 0,C 0,E1 0.1598,E2 90.072} C_DIS
LIN {X 1.0484,Y 4.6368,Z 1,A -2.6018,B 0,C 0,E1 0.1598,E2 90.072} C_DIS
LIN {X 1.5562,Y 4.491,Z 1,A -2.5893,B 0,C 0,E1 0.1598,E2 90.0721} C_DIS
LIN {X 2.0449,Y 4.2903,Z 1,A -2.5797,B 0,C 0,E1 0.1598,E2 90.0721} C_DIS
LIN {X 2.5089,Y 4.0375,Z 1,A -2.5733,B 0,C 0,E1 0.1598,E2 90.0721} C_DIS
LIN {X 2.9418,Y 3.7347,Z 1,A -2.5701,B 0,C 0,E1 0.1598,E2 90.0721} C_DIS
LIN {X 3.3377,Y 3.3849,Z 1,A -2.5702,B 0,C 0,E1 0.1598,E2 90.0721} C_DIS
LIN {X 3.6924,Y 2.9933,Z 1,A -2.5737,B 0,C 0,E1 0.1598,E2 90.0721} C_DIS
LIN {X 4.0022,Y 2.5654,Z 1,A -2.5804,B 0,C 0,E1 0.1598,E2 90.0721} C_DIS
LIN {X 4.2618,Y 2.1052,Z 1,A -2.5903,B 0,C 0,E1 0.1598,E2 90.072} C_DIS
LIN {X 4.4689,Y 1.6192,Z 1,A -2.6032,B 0,C 0,E1 0.1598,E2 90.072} C_DIS
LIN {X 4.6203,Y 1.113,Z 1,A -2.619,B 0,C 0,E1 0.1598,E2 90.072} C_DIS
LIN {X 4.717,Y 0.5936,Z 1,A -2.6374,B 0,C 0,E1 0.1598,E2 90.072} C_DIS
LIN {X 4.7528,Y 0.0665,Z 1,A -2.6584,B 0,C 0,E1 0.1598,E2 90.0719} C_DIS
LIN {X 4.73,Y -0.4613,Z 1,A -2.6816,B 0,C 0,E1 0.1598,E2 90.0719} C_DIS
LIN {X 4.6507,Y -0.9836,Z 1,A -2.7066,B 0,C 0,E1 0.1598,E2 90.0719} C_DIS
LIN {X 4.5132,Y -1.4937,Z 1,A -2.7333,B 0,C 0,E1 0.1598,E2 90.0718} C_DIS
LIN {X 4.3187,Y -1.9849,Z 1,A -2.7612,B 0,C 0,E1 0.1598,E2 90.0718} C_DIS
LIN {X 4.0716,Y -2.4519,Z 1,A -2.7901,B 0,C 0,E1 0.1598,E2 90.0718} C_DIS
LIN {X 3.7751,Y -2.8892,Z 1,A -2.8195,B 0,C 0,E1 0.1598,E2 90.0718} C_DIS
LIN {X 3.4318,Y -3.2907,Z 1,A -2.8492,B 0,C 0,E1 0.1598,E2 90.0717} C_DIS
LIN {X 3.0436,Y -3.6491,Z 1,A -2.8786,B 0,C 0,E1 0.1598,E2 90.0717} C_DIS
LIN {X 2.6193,Y -3.9638,Z 1,A -2.9075,B 0,C 0,E1 0.1598,E2 90.0717} C_DIS
LIN {X 2.1632,Y -4.23,Z 1,A -2.9356,B 0,C 0,E1 0.1598,E2 90.0717} C_DIS
LIN {X 1.6804,Y -4.4443,Z 1,A -2.9624,B 0,C 0,E1 0.1598,E2 90.0717} C_DIS
LIN {X 1.1767,Y -4.6035,Z 1,A -2.9876,B 0,C 0,E1 0.1598,E2 90.0716} C_DIS
LIN {X 0.6585,Y -4.7065,Z 1,A -3.011,B 0,C 0,E1 0.1598,E2 90.0716} C_DIS
LIN {X 0.0001,Y -4.7537,Z 1,A -3.0372,B 0,C 0,E1 0.1598,E2 90.0716} C_DIS
Enddeposition()
LIN {X 0.0001,Y -4.7537,Z 1,A -3.0372,B 0,C 0,E1 0.1598,E2 90.0716} C_DIS
Startdeposition()
$VEL.CP = VEL_PRINT
LIN {X 0.62,Y -5.6505,Z 1,A -3.0519,B 0,C 0,E1 0.1598,E2 90.0709} C_DIS
LIN {X 1.4007,Y -5.5096,Z 1,A -3.0178,B 0,C 0,E1 0.1598,E2 90.0715} C_DIS
LIN {X 2.1538,Y -5.2601,Z 1,A -2.9796,B 0,C 0,E1 0.1598,E2 90.0715} C_DIS
LIN {X 2.865,Y -4.9088,Z 1,A -2.9386,B 0,C 0,E1 0.1598,E2 90.0716} C_DIS
LIN {X 3.5219,Y -4.4641,Z 1,A -2.8956,B 0,C 0,E1 0.1598,E2 90.0716} C_DIS
LIN {X 4.1076,Y -3.9289,Z 1,A -2.8514,B 0,C 0,E1 0.1598,E2 90.0716} C_DIS
LIN {X 4.6149,Y -3.3191,Z 1,A -2.8069,B 0,C 0,E1 0.1598,E2 90.0716} C_DIS
LIN {X 5.0319,Y -2.6443,Z 1,A -2.7629,B 0,C 0,E1 0.1598,E2 90.0716} C_DIS
LIN {X 5.351,Y -1.918,Z 1,A -2.7204,B 0,C 0,E1 0.1598,E2 90.0716} C_DIS
LIN {X 5.5671,Y -1.1546,Z 1,A -2.68,B 0,C 0,E1 0.1598,E2 90.0716} C_DIS
LIN {X 5.6721,Y -0.3684,Z 1,A -2.6429,B 0,C 0,E1 0.1598,E2 90.0717} C_DIS
LIN {X 5.6686,Y 0.4249,Z 1,A -2.6094,B 0,C 0,E1 0.1598,E2 90.0717} C_DIS
LIN {X 5.5539,Y 1.2098,Z 1,A -2.5804,B 0,C 0,E1 0.1598,E2 90.0717} C_DIS
LIN {X 5.3319,Y 1.9714,Z 1,A -2.5563,B 0,C 0,E1 0.1598,E2 90.0718} C_DIS
LIN {X 4.9138,Y 2.8708,Z 1,A -2.5334,B 0,C 0,E1 0.1598,E2 90.0717} C_DIS
LIN {X 4.1914,Y 3.8403,Z 1,A -2.519,B 0,C 0,E1 0.1598,E2 90.0717} C_DIS
LIN {X 3.5797,Y 4.4163,Z 1,A -2.5176,B 0,C 0,E1 0.1598,E2 90.072} C_DIS
LIN {X 2.8901,Y 4.8963,Z 1,A -2.5228,B 0,C 0,E1 0.1598,E2 90.072} C_DIS
LIN {X 2.1364,Y 5.2681,Z 1,A -2.5349,B 0,C 0,E1 0.1598,E2 90.0721} C_DIS
LIN {X 1.3364,Y 5.5247,Z 1,A -2.5537,B 0,C 0,E1 0.1598,E2 90.0721} C_DIS
LIN {X 0.5077,Y 5.6611,Z 1,A -2.5785,B 0,C 0,E1 0.1598,E2 90.0721} C_DIS
LIN {X -0.3325,Y 5.676,Z 1,A -2.6089,B 0,C 0,E1 0.1598,E2 90.0721} C_DIS
LIN {X -1.2513,Y 5.5498,Z 1,A -2.6481,B 0,C 0,E1 0.1598,E2 90.0721} C_DIS
LIN {X -1.9393,Y 5.3432,Z 1,A -2.6822,B 0,C 0,E1 0.1598,E2 90.072} C_DIS
LIN {X -2.6716,Y 5.0236,Z 1,A -2.7226,B 0,C 0,E1 0.1598,E2 90.0719} C_DIS
LIN {X -3.4724,Y 4.4979,Z 1,A -2.7742,B 0,C 0,E1 0.1598,E2 90.0718} C_DIS
LIN {X -4.0465,Y 3.9904,Z 1,A -2.8167,B 0,C 0,E1 0.1598,E2 90.0717} C_DIS
LIN {X -4.5461,Y 3.4095,Z 1,A -2.8595,B 0,C 0,E1 0.1598,E2 90.0716} C_DIS
LIN {X -5.0613,Y 2.6016,Z 1,A -2.9123,B 0,C 0,E1 0.1598,E2 90.0713} C_DIS
LIN {X -5.5056,Y 1.4349,Z 1,A -2.9773,B 0,C 0,E1 0.1598,E2 90.0708} C_DIS
LIN {X -5.6786,Y 0.3563,Z 1,A -3.0293,B 0,C 0,E1 0.1598,E2 90.071} C_DIS
LIN {X -5.6398,Y -0.7607,Z 1,A -3.0748,B 0,C 0,E1 0.1598,E2 90.0708} C_DIS
LIN {X -5.3577,Y -1.9044,Z 1,A -3.1125,B 0,C 0,E1 0.1598,E2 90.0708} C_DIS
LIN {X -5.0565,Y -2.5997,Z 1,A -3.1311,B 0,C 0,E1 0.1598,E2 90.0711} C_DIS
LIN {X -4.6654,Y -3.2488,Z 1,A -3.1441,B 0,C 0,E1 0.1598,E2 90.0711} C_DIS
LIN {X -4.1925,Y -3.8411,Z 1,A -3.1518,B 0,C 0,E1 0.1598,E2 90.0711} C_DIS
LIN {X -3.6427,Y -4.3626,Z 1,A -3.1536,B 0,C 0,E1 0.1598,E2 90.0712} C_DIS
LIN {X -3.0314,Y -4.8101,Z 1,A -3.1501,B 0,C 0,E1 0.1598,E2 90.0712} C_DIS
LIN {X -2.3642,Y -5.1694,Z 1,A -3.1408,B 0,C 0,E1 0.1598,E2 90.0713} C_DIS
LIN {X -1.6553,Y -5.4366,Z 1,A -3.1261,B 0,C 0,E1 0.1598,E2 90.0713} C_DIS
LIN {X -0.9178,Y -5.6096,Z 1,A -3.1063,B 0,C 0,E1 0.1598,E2 90.0714} C_DIS
LIN {X 0.0259,Y -5.6891,Z 1,A -3.0751,B 0,C 0,E1 0.1598,E2 90.0714} C_DIS
Enddeposition()
LIN {X 0.0259,Y -5.6891,Z 1,A -3.0751,B 0,C 0,E1 0.1598,E2 90.0714} C_DIS
Startdeposition()
$VEL.CP = VEL_PRINT
LIN {X -0.4859,Y -6.6021,Z 1,A -3.1321,B 0,C 0,E1 0.1598,E2 90.0708} C_DIS
LIN {X -1.1513,Y -6.5191,Z 1,A -3.1535,B 0,C 0,E1 0.1598,E2 90.0713} C_DIS
LIN {X -1.8046,Y -6.3678,Z 1,A -3.1711,B 0,C 0,E1 0.1598,E2 90.0713} C_DIS
LIN {X -2.4403,Y -6.154,Z 1,A -3.1854,B 0,C 0,E1 0.1598,E2 90.0713} C_DIS
LIN {X -3.0501,Y -5.8747,Z 1,A -3.1959,B 0,C 0,E1 0.1598,E2 90.0713} C_DIS
LIN {X -3.6289,Y -5.5362,Z 1,A -3.2029,B 0,C 0,E1 0.1598,E2 90.0713} C_DIS
LIN {X -4.1711,Y -5.1415,Z 1,A -3.2061,B 0,C 0,E1 0.1598,E2 90.0713} C_DIS
LIN {X -4.6697,Y -4.6931,Z 1,A -3.2055,B 0,C 0,E1 0.1598,E2 90.0712} C_DIS
LIN {X -5.1195,Y -4.1956,Z 1,A -3.201,B 0,C 0,E1 0.1598,E2 90.0712} C_DIS
LIN {X -5.5179,Y -3.6563,Z 1,A -3.1929,B 0,C 0,E1 0.1598,E2 90.0712} C_DIS
LIN {X -5.8607,Y -3.0799,Z 1,A -3.1812,B 0,C 0,E1 0.1598,E2 90.0712} C_DIS
LIN {X -6.1422,Y -2.4713,Z 1,A -3.1659,B 0,C 0,E1 0.1598,E2 90.0712} C_DIS
LIN {X -6.3608,Y -1.8373,Z 1,A -3.1472,B 0,C 0,E1 0.1598,E2 90.0712} C_DIS
LIN {X -6.5135,Y -1.1842,Z 1,A -3.1253,B 0,C 0,E1 0.1598,E2 90.0712} C_DIS
LIN {X -6.5994,Y -0.5193,Z 1,A -3.1005,B 0,C 0,E1 0.1598,E2 90.0712} C_DIS
LIN {X -6.6185,Y 0.1512,Z 1,A -3.073,B 0,C 0,E1 0.1598,E2 90.0712} C_DIS
LIN {X -6.5705,Y 0.8201,Z 1,A -3.0431,B 0,C 0,E1 0.1598,E2 90.0712} C_DIS
LIN {X -6.4533,Y 1.4804,Z 1,A -3.011,B 0,C 0,E1 0.1598,E2 90.0713} C_DIS
LIN {X -6.2703,Y 2.1256,Z 1,A -2.9772,B 0,C 0,E1 0.1598,E2 90.0713} C_DIS
LIN {X -6.0231,Y 2.749,Z 1,A -2.9418,B 0,C 0,E1 0.1598,E2 90.0715} C_DIS
LIN {X -5.7138,Y 3.3439,Z 1,A -2.9054,B 0,C 0,E1 0.1598,E2 90.0715} C_DIS
LIN {X -5.3465,Y 3.905,Z 1,A -2.8683,B 0,C 0,E1 0.1598,E2 90.0715} C_DIS
LIN {X -4.923,Y 4.4251,Z 1,A -2.8309,B 0,C 0,E1 0.1598,E2 90.0717} C_DIS
LIN {X -4.4502,Y 4.9005,Z 1,A -2.7935,B 0,C 0,E1 0.1598,E2 90.0717} C_DIS
LIN {X -3.9313,Y 5.3254,Z 1,A -2.7565,B 0,C 0,E1 0.1598,E2 90.0718} C_DIS
LIN {X -3.3731,Y 5.697,Z 1,A -2.7203,B 0,C 0,E1 0.1598,E2 90.0718} C_DIS
LIN {X -2.7796,Y 6.0092,Z 1,A -2.6853,B 0,C 0,E1 0.1598,E2 90.0719} C_DIS
LIN {X -2.1575,Y 6.2596,Z 1,A -2.6518,B 0,C 0,E1 0.1598,E2 90.072} C_DIS
LIN {X -1.5133,Y 6.4457,Z 1,A -2.6202,B 0,C 0,E1 0.1598,E2 90.072} C_DIS
LIN {X -0.8535,Y 6.566,Z 1,A -2.5908,B 0,C 0,E1 0.1598,E2 90.0721} C_DIS
LIN {X -0.1848,Y 6.6163,Z 1,A -2.564,B 0,C 0,E1 0.1598,E2 90.0721} C_DIS
LIN {X 0.4857,Y 6.6026,Z 1,A -2.5398,B 0,C 0,E1 0.1598,E2 90.0721} C_DIS
LIN {X 1.1512,Y 6.5202,Z 1,A -2.5187,B 0,C 0,E1 0.1598,E2 90.0722} C_DIS
LIN {X 1.8048,Y 6.3701,Z 1,A -2.5009,B 0,C 0,E1 0.1598,E2 90.0722} C_DIS
LIN {X 2.4399,Y 6.1548,Z 1,A -2.4866,B 0,C 0,E1 0.1598,E2 90.0722} C_DIS
LIN {X 3.05,Y 5.8763,Z 1,A -2.4758,B 0,C 0,E1 0.1598,E2 90.0722} C_DIS
LIN {X 3.6285,Y 5.5369,Z 1,A -2.4687,B 0,C 0,E1 0.1598,E2 90.0722} C_DIS
LIN {X 4.1699,Y 5.1411,Z 1,A -2.4655,B 0,C 0,E1 0.1598,E2 90.0722} C_DIS
LIN {X 4.6692,Y 4.6936,Z 1,A -2.466,B 0,C 0,E1 0.1598,E2 90.0722} C_DIS
LIN {X 5.1202,Y 4.1973,Z 1,A -2.4703,B 0,C 0,E1 0.1598,E2 90.0722} C_DIS
LIN {X 5.5178,Y 3.6572,Z 1,A -2.4785,B 0,C 0,E1 0.1598,E2 90.0721} C_DIS
LIN {X 5.8603,Y 3.0807,Z 1,A -2.4902,B 0,C 0,E1 0.1598,E2 90.0721} C_DIS
LIN {X 6.141,Y 2.4717,Z 1,A -2.5056,B 0,C 0,E1 0.1598,E2 90.0721} C_DIS
LIN {X 6.3595,Y 1.8376,Z 1,A -2.5244,B 0,C 0,E1 0.1598,E2 90.072} C_DIS
LIN {X 6.5123,Y 1.1846,Z 1,A -2.5464,B 0,C 0,E1 0.1598,E2 90.072} C_DIS
LIN {X 6.5997,Y 0.5197,Z 1,A -2.5714,B 0,C 0,E1 0.1598,E2 90.0719} C_DIS
LIN {X 6.6205,Y -0.1506,Z 1,A -2.599,B 0,C 0,E1 0.1598,E2 90.0719} C_DIS
LIN {X 6.5706,Y -0.8195,Z 1,A -2.6292,B 0,C 0,E1 0.1598,E2 90.0719} C_DIS
LIN {X 6.4534,Y -1.4798,Z 1,A -2.6615,B 0,C 0,E1 0.1598,E2 90.0718} C_DIS
LIN {X 6.2705,Y -2.125,Z 1,A -2.6956,B 0,C 0,E1 0.1598,E2 90.0718} C_DIS
LIN {X 6.0233,Y -2.7484,Z 1,A -2.7311,B 0,C 0,E1 0.1598,E2 90.0718} C_DIS
LIN {X 5.7138,Y -3.3434,Z 1,A -2.7677,B 0,C 0,E1 0.1598,E2 90.0718} C_DIS
LIN {X 5.3455,Y -3.904,Z 1,A -2.805,B 0,C 0,E1 0.1598,E2 90.0717} C_DIS
LIN {X 4.9232,Y -4.425,Z 1,A -2.8426,B 0,C 0,E1 0.1598,E2 90.0717} C_DIS
LIN {X 4.45,Y -4.9001,Z 1,A -2.8802,B 0,C 0,E1 0.1598,E2 90.0717} C_DIS
LIN {X 3.9316,Y -5.3255,Z 1,A -2.9172,B 0,C 0,E1 0.1598,E2 90.0716} C_DIS
LIN {X 3.3734,Y -5.6971,Z 1,A -2.9535,B 0,C 0,E1 0.1598,E2 90.0716} C_DIS
LIN {X 2.7791,Y -6.0078,Z 1,A -2.9885,B 0,C 0,E1 0.1598,E2 90.0716} C_DIS
LIN {X 2.1573,Y -6.259,Z 1,A -3.022,B 0,C 0,E1 0.1598,E2 90.0716} C_DIS
LIN {X 1.5127,Y -6.4445,Z 1,A -3.0535,B 0,C 0,E1 0.1598,E2 90.0715} C_DIS
LIN {X 0.8533,Y -6.566,Z 1,A -3.0828,B 0,C 0,E1 0.1598,E2 90.0715} C_DIS
LIN {X 0.0169,Y -6.6225,Z 1,A -3.1159,B 0,C 0,E1 0.1598,E2 90.0715} C_DIS
Enddeposition()
LIN {X 0.0169,Y -6.6225,Z 1,A -3.1159,B 0,C 0,E1 0.1598,E2 90.0715} C_DIS
Startdeposition()
$VEL.CP = VEL_PRINT
LIN {X 0.2384,Y -7.5535,Z 1,A -3.1468,B 0,C 0,E1 0.1598,E2 90.0708} C_DIS
LIN {X 1.3624,Y -7.4302,Z 1,A -3.1008,B 0,C 0,E1 0.1598,E2 90.0714} C_DIS
LIN {X 2.1091,Y -7.2529,Z 1,A -3.066,B 0,C 0,E1 0.1598,E2 90.0714} C_DIS
LIN {X 3.1484,Y -6.8715,Z 1,A -3.0116,B 0,C 0,E1 0.1598,E2 90.0714} C_DIS
LIN {X 4.0754,Y -6.3591,Z 1,A -2.9559,B 0,C 0,E1 0.1598,E2 90.0715} C_DIS
LIN {X 4.7616,Y -5.8621,Z 1,A -2.9096,B 0,C 0,E1 0.1598,E2 90.0715} C_DIS
LIN {X 5.3881,Y -5.2918,Z 1,A -2.8624,B 0,C 0,E1 0.1598,E2 90.0715} C_DIS
LIN {X 6.1273,Y -4.425,Z 1,A -2.7983,B 0,C 0,E1 0.1598,E2 90.0715} C_DIS
LIN {X 6.5954,Y -3.6789,Z 1,A -2.7496,B 0,C 0,E1 0.1598,E2 90.0716} C_DIS
LIN {X 7.0592,Y -2.6978,Z 1,A -2.6907,B 0,C 0,E1 0.1598,E2 90.0715} C_DIS
LIN {X 7.3559,Y -1.712,Z 1,A -2.638,B 0,C 0,E1 0.1598,E2 90.0715} C_DIS
LIN {X 7.5262,Y -0.6969,Z 1,A -2.5885,B 0,C 0,E1 0.1598,E2 90.0715} C_DIS
LIN {X 7.5359,Y 0.5664,Z 1,A -2.5342,B 0,C 0,E1 0.1598,E2 90.0712} C_DIS
LIN {X 7.3457,Y 1.7584,Z 1,A -2.4908,B 0,C 0,E1 0.1598,E2 90.0714} C_DIS
LIN {X 7.1324,Y 2.4987,Z 1,A -2.4677,B 0,C 0,E1 0.1598,E2 90.0718} C_DIS
LIN {X 6.731,Y 3.4376,Z 1,A -2.4427,B 0,C 0,E1 0.1598,E2 90.0718} C_DIS
LIN {X 6.1837,Y 4.3388,Z 1,A -2.4247,B 0,C 0,E1 0.1598,E2 90.0718} C_DIS
LIN {X 5.6476,Y 5.0224,Z 1,A -2.4157,B 0,C 0,E1 0.1598,E2 90.072} C_DIS
LIN {X 4.8286,Y 5.8087,Z 1,A -2.4126,B 0,C 0,E1 0.1598,E2 90.072} C_DIS
LIN {X 4.0774,Y 6.3632,Z 1,A -2.4171,B 0,C 0,E1 0.1598,E2 90.0721} C_DIS
LIN {X 3.2504,Y 6.8219,Z 1,A -2.4283,B 0,C 0,E1 0.1598,E2 90.0722} C_DIS
LIN {X 2.4265,Y 7.1584,Z 1,A -2.4446,B 0,C 0,E1 0.1598,E2 90.0722} C_DIS
LIN {X 1.2876,Y 7.4432,Z 1,A -2.4746,B 0,C 0,E1 0.1598,E2 90.0722} C_DIS
LIN {X 0.0592,Y 7.5575,Z 1,A -2.5152,B 0,C 0,E1 0.1598,E2 90.0722} C_DIS
LIN {X -1.1059,Y 7.4713,Z 1,A -2.5618,B 0,C 0,E1 0.1598,E2 90.0722} C_DIS
LIN {X -1.9222,Y 7.3038,Z 1,A -2.599,B 0,C 0,E1 0.1598,E2 90.0721} C_DIS
LIN {X -2.715,Y 7.047,Z 1,A -2.6391,B 0,C 0,E1 0.1598,E2 90.0721} C_DIS
LIN {X -3.4751,Y 6.7055,Z 1,A -2.6815,B 0,C 0,E1 0.1598,E2 90.0719} C_DIS
LIN {X -4.4898,Y 6.0798,Z 1,A -2.7451,B 0,C 0,E1 0.1598,E2 90.0717} C_DIS
LIN {X -5.0999,Y 5.5776,Z 1,A -2.7888,B 0,C 0,E1 0.1598,E2 90.0717} C_DIS
LIN {X -5.8053,Y 4.8311,Z 1,A -2.8461,B 0,C 0,E1 0.1598,E2 90.0715} C_DIS
LIN {X -6.2962,Y 4.1723,Z 1,A -2.8919,B 0,C 0,E1 0.1598,E2 90.0715} C_DIS
LIN {X -6.807,Y 3.2812,Z 1,A -2.9479,B 0,C 0,E1 0.1598,E2 90.0712} C_DIS
LIN {X -7.2489,Y 2.1212,Z 1,A -3.0127,B 0,C 0,E1 0.1598,E2 90.0709} C_DIS
LIN {X -7.4456,Y 1.2717,Z 1,A -3.0559,B 0,C 0,E1 0.1598,E2 90.0711} C_DIS
LIN {X -7.5562,Y 0.1201,Z 1,A -3.1082,B 0,C 0,E1 0.1598,E2 90.0708} C_DIS
LIN {X -7.5248,Y -0.7097,Z 1,A -3.1422,B 0,C 0,E1 0.1598,E2 90.0711} C_DIS
LIN {X -7.3086,Y -1.9203,Z 1,A -3.1848,B 0,C 0,E1 0.1598,E2 90.0706} C_DIS
LIN {X -6.9997,Y -2.8486,Z 1,A -3.2126,B 0,C 0,E1 0.1598,E2 90.0708} C_DIS
LIN {X -6.5598,Y -3.7438,Z 1,A -3.2343,B 0,C 0,E1 0.1598,E2 90.0708} C_DIS
LIN {X -6.1272,Y -4.4144,Z 1,A -3.2468,B 0,C 0,E1 0.1598,E2 90.071} C_DIS
LIN {X -5.3827,Y -5.3052,Z 1,A -3.2568,B 0,C 0,E1 0.1598,E2 90.0708} C_DIS
LIN {X -4.5636,Y -6.023,Z 1,A -3.2571,B 0,C 0,E1 0.1598,E2 90.071} C_DIS
LIN {X -3.5199,Y -6.688,Z 1,A -3.2469,B 0,C 0,E1 0.1598,E2 90.071} C_DIS
LIN {X -2.3983,Y -7.1625,Z 1,A -3.2259,B 0,C 0,E1 0.1598,E2 90.0711} C_DIS
LIN {X -1.6589,Y -7.3732,Z 1,A -3.2078,B 0,C 0,E1 0.1598,E2 90.0713} C_DIS
LIN {X -0.8228,Y -7.5079,Z 1,A -3.1829,B 0,C 0,E1 0.1598,E2 90.0713} C_DIS
LIN {X 0.0226,Y -7.5548,Z 1,A -3.1539,B 0,C 0,E1 0.1598,E2 90.0713} C_DIS
Enddeposition()
LIN {X 0.0226,Y -7.5548,Z 1,A -3.1539,B 0,C 0,E1 0.1598,E2 90.0713} C_DIS
Startdeposition()
$VEL.CP = VEL_PRINT
LIN {X -0.5223,Y -8.472,Z 1,A -3.2123,B 0,C 0,E1 0.1598,E2 90.0707} C_DIS
LIN {X -1.2769,Y -8.39,Z 1,A -3.237,B 0,C 0,E1 0.1598,E2 90.0712} C_DIS
LIN {X -2.0214,Y -8.2421,Z 1,A -3.2581,B 0,C 0,E1 0.1598,E2 90.0712} C_DIS
LIN {X -2.7498,Y -8.0287,Z 1,A -3.2757,B 0,C 0,E1 0.1598,E2 90.0712} C_DIS
LIN {X -3.4567,Y -7.7522,Z 1,A -3.29,B 0,C 0,E1 0.1598,E2 90.0712} C_DIS
LIN {X -4.1354,Y -7.412,Z 1,A -3.3005,B 0,C 0,E1 0.1598,E2 90.0712} C_DIS
LIN {X -4.7808,Y -7.0123,Z 1,A -3.3072,B 0,C 0,E1 0.1598,E2 90.0711} C_DIS
LIN {X -5.5355,Y -6.4373,Z 1,A -3.3106,B 0,C 0,E1 0.1598,E2 90.071} C_DIS
LIN {X -6.3159,Y -5.6768,Z 1,A -3.307,B 0,C 0,E1 0.1598,E2 90.0708} C_DIS
LIN {X -7.0633,Y -4.7127,Z 1,A -3.2937,B 0,C 0,E1 0.1598,E2 90.0708} C_DIS
LIN {X -7.5131,Y -3.957,Z 1,A -3.2786,B 0,C 0,E1 0.1598,E2 90.0709} C_DIS
LIN {X -8.0118,Y -2.7993,Z 1,A -3.2478,B 0,C 0,E1 0.1598,E2 90.0706} C_DIS
LIN {X -8.2485,Y -1.9943,Z 1,A -3.223,B 0,C 0,E1 0.1598,E2 90.0709} C_DIS
LIN {X -8.4053,Y -1.1701,Z 1,A -3.1941,B 0,C 0,E1 0.1598,E2 90.0709} C_DIS
LIN {X -8.4804,Y -0.3344,Z 1,A -3.1617,B 0,C 0,E1 0.1598,E2 90.071} C_DIS
LIN {X -8.4724,Y 0.5044,Z 1,A -3.1262,B 0,C 0,E1 0.1598,E2 90.071} C_DIS
LIN {X -8.3803,Y 1.3383,Z 1,A -3.0878,B 0,C 0,E1 0.1598,E2 90.0711} C_DIS
LIN {X -8.2067,Y 2.1592,Z 1,A -3.0469,B 0,C 0,E1 0.1598,E2 90.0711} C_DIS
LIN {X -7.9534,Y 2.959,Z 1,A -3.004,B 0,C 0,E1 0.1598,E2 90.0713} C_DIS
LIN {X -7.6225,Y 3.7299,Z 1,A -2.9594,B 0,C 0,E1 0.1598,E2 90.0713} C_DIS
LIN {X -7.1095,Y 4.6447,Z 1,A -2.9019,B 0,C 0,E1 0.1598,E2 90.0713} C_DIS
LIN {X -6.4348,Y 5.5374,Z 1,A -2.8396,B 0,C 0,E1 0.1598,E2 90.0713} C_DIS
LIN {X -5.8669,Y 6.135,Z 1,A -2.7938,B 0,C 0,E1 0.1598,E2 90.0717} C_DIS
LIN {X -5.2439,Y 6.6751,Z 1,A -2.7481,B 0,C 0,E1 0.1598,E2 90.0717} C_DIS
LIN {X -4.5712,Y 7.1517,Z 1,A -2.7033,B 0,C 0,E1 0.1598,E2 90.0719} C_DIS
LIN {X -3.8555,Y 7.561,Z 1,A -2.6597,B 0,C 0,E1 0.1598,E2 90.0719} C_DIS
LIN {X -3.1037,Y 7.8992,Z 1,A -2.6177,B 0,C 0,E1 0.1598,E2 90.072} C_DIS
LIN {X -2.3226,Y 8.163,Z 1,A -2.5778,B 0,C 0,E1 0.1598,E2 90.0721} C_DIS
LIN {X -1.5197,Y 8.3502,Z 1,A -2.5403,B 0,C 0,E1 0.1598,E2 90.0721} C_DIS
LIN {X -0.7024,Y 8.4583,Z 1,A -2.5056,B 0,C 0,E1 0.1598,E2 90.0722} C_DIS
LIN {X 0.1214,Y 8.4872,Z 1,A -2.4739,B 0,C 0,E1 0.1598,E2 90.0722} C_DIS
LIN {X 0.9441,Y 8.4346,Z 1,A -2.4457,B 0,C 0,E1 0.1598,E2 90.0723} C_DIS
LIN {X 1.7577,Y 8.3025,Z 1,A -2.4212,B 0,C 0,E1 0.1598,E2 90.0723} C_DIS
LIN {X 2.5548,Y 8.0923,Z 1,A -2.4007,B 0,C 0,E1 0.1598,E2 90.0723} C_DIS
LIN {X 3.3278,Y 7.8061,Z 1,A -2.3842,B 0,C 0,E1 0.1598,E2 90.0723} C_DIS
LIN {X 4.2522,Y 7.3507,Z 1,A -2.3692,B 0,C 0,E1 0.1598,E2 90.0723} C_DIS
LIN {X 4.9716,Y 6.8844,Z 1,A -2.3623,B 0,C 0,E1 0.1598,E2 90.0723} C_DIS
LIN {X 5.8407,Y 6.161,Z 1,A -2.3606,B 0,C 0,E1 0.1598,E2 90.0721} C_DIS
LIN {X 6.4077,Y 5.568,Z 1,A -2.3649,B 0,C 0,E1 0.1598,E2 90.0721} C_DIS
LIN {X 6.9146,Y 4.9228,Z 1,A -2.3735,B 0,C 0,E1 0.1598,E2 90.0721} C_DIS
LIN {X 7.357,Y 4.2318,Z 1,A -2.3864,B 0,C 0,E1 0.1598,E2 90.0721} C_DIS
LIN {X 7.7308,Y 3.5015,Z 1,A -2.4035,B 0,C 0,E1 0.1598,E2 90.0721} C_DIS
LIN {X 8.0324,Y 2.7386,Z 1,A -2.4247,B 0,C 0,E1 0.1598,E2 90.0721} C_DIS
LIN {X 8.2595,Y 1.9503,Z 1,A -2.4497,B 0,C 0,E1 0.1598,E2 90.072} C_DIS
LIN {X 8.4094,Y 1.1437,Z 1,A -2.4784,B 0,C 0,E1 0.1598,E2 90.072} C_DIS
LIN {X 8.4811,Y 0.3265,Z 1,A -2.5104,B 0,C 0,E1 0.1598,E2 90.0719} C_DIS
LIN {X 8.4737,Y -0.4938,Z 1,A -2.5455,B 0,C 0,E1 0.1598,E2 90.0719} C_DIS
LIN {X 8.3854,Y -1.3094,Z 1,A -2.5833,B 0,C 0,E1 0.1598,E2 90.0718} C_DIS
LIN {X 8.2192,Y -2.1127,Z 1,A -2.6236,B 0,C 0,E1 0.1598,E2 90.0718} C_DIS
LIN {X 7.9765,Y -2.8963,Z 1,A -2.6657,B 0,C 0,E1 0.1598,E2 90.0717} C_DIS
LIN {X 7.6596,Y -3.6529,Z 1,A -2.7095,B 0,C 0,E1 0.1598,E2 90.0717} C_DIS
LIN {X 7.0616,Y -4.7151,Z 1,A -2.7763,B 0,C 0,E1 0.1598,E2 90.0713} C_DIS
LIN {X 6.4426,Y -5.5278,Z 1,A -2.8337,B 0,C 0,E1 0.1598,E2 90.0715} C_DIS
LIN {X 5.881,Y -6.1217,Z 1,A -2.8797,B 0,C 0,E1 0.1598,E2 90.0715} C_DIS
LIN {X 5.2645,Y -6.6581,Z 1,A -2.9251,B 0,C 0,E1 0.1598,E2 90.0715} C_DIS
LIN {X 4.3245,Y -7.3079,Z 1,A -2.9871,B 0,C 0,E1 0.1598,E2 90.0715} C_DIS
LIN {X 3.2458,Y -7.8456,Z 1,A -3.0495,B 0,C 0,E1 0.1598,E2 90.0714} C_DIS
LIN {X 2.2755,Y -8.1772,Z 1,A -3.0992,B 0,C 0,E1 0.1598,E2 90.0714} C_DIS
LIN {X 1.4754,Y -8.3587,Z 1,A -3.1362,B 0,C 0,E1 0.1598,E2 90.0714} C_DIS
LIN {X 0.6616,Y -8.4625,Z 1,A -3.1704,B 0,C 0,E1 0.1598,E2 90.0714} C_DIS
LIN {X 0.6616,Y -8.4625,Z 1,A -3.1704,B 0,C 0,E1 0.1598,E2 90.0714} C_DIS
Enddeposition()
LIN {X 0.0001,Y -4.7539,Z 2,A -3.0223,B 0,C 0,E1 0.1598,E2 90.0603} C_DIS
Startdeposition()
$VEL.CP = VEL_PRINT
LIN {X 0.0001,Y -4.7539,Z 2,A -3.028,B 0,C 0,E1 0.1598,E2 90.066} C_DIS
LIN {X 0.6703,Y -4.7046,Z 2,A -3.0061,B 0,C 0,E1 0.1598,E2 90.0709} C_DIS
LIN {X 1.1975,Y -4.5981,Z 2,A -2.9829,B 0,C 0,E1 0.1598,E2 90.0716} C_DIS
LIN {X 1.7094,Y -4.4335,Z 2,A -2.9572,B 0,C 0,E1 0.1598,E2 90.0716} C_DIS
LIN {X 2.199,Y -4.2112,Z 2,A -2.9298,B 0,C 0,E1 0.1598,E2 90.0716} C_DIS
LIN {X 2.6609,Y -3.9362,Z 2,A -2.9011,B 0,C 0,E1 0.1598,E2 90.0716} C_DIS
LIN {X 3.0897,Y -3.6114,Z 2,A -2.8716,B 0,C 0,E1 0.1598,E2 90.0716} C_DIS
LIN {X 3.479,Y -3.2404,Z 2,A -2.8416,B 0,C 0,E1 0.1598,E2 90.0717} C_DIS
LIN {X 3.8218,Y -2.826,Z 2,A -2.8114,B 0,C 0,E1 0.1598,E2 90.0717} C_DIS
LIN {X 4.1168,Y -2.3763,Z 2,A -2.7815,B 0,C 0,E1 0.1598,E2 90.0717} C_DIS
LIN {X 4.359,Y -1.8961,Z 2,A -2.7523,B 0,C 0,E1 0.1598,E2 90.0717} C_DIS
LIN {X 4.5445,Y -1.3913,Z 2,A -2.7241,B 0,C 0,E1 0.1598,E2 90.0718} C_DIS
LIN {X 4.6732,Y -0.8691,Z 2,A -2.6972,B 0,C 0,E1 0.1598,E2 90.0718} C_DIS
LIN {X 4.7428,Y -0.3358,Z 2,A -2.672,B 0,C 0,E1 0.1598,E2 90.0718} C_DIS
LIN {X 4.7477,Y 0.202,Z 2,A -2.6491,B 0,C 0,E1 0.1598,E2 90.0718} C_DIS
LIN {X 4.6956,Y 0.7371,Z 2,A -2.6284,B 0,C 0,E1 0.1598,E2 90.0719} C_DIS
LIN {X 4.5829,Y 1.263,Z 2,A -2.6102,B 0,C 0,E1 0.1598,E2 90.0719} C_DIS
LIN {X 4.41,Y 1.7723,Z 2,A -2.5951,B 0,C 0,E1 0.1598,E2 90.0719} C_DIS
LIN {X 4.1815,Y 2.2592,Z 2,A -2.5829,B 0,C 0,E1 0.1598,E2 90.0719} C_DIS
LIN {X 3.9004,Y 2.7176,Z 2,A -2.5739,B 0,C 0,E1 0.1598,E2 90.072} C_DIS
LIN {X 3.5682,Y 3.1405,Z 2,A -2.5682,B 0,C 0,E1 0.1598,E2 90.072} C_DIS
LIN {X 3.1898,Y 3.5228,Z 2,A -2.566,B 0,C 0,E1 0.1598,E2 90.072} C_DIS
LIN {X 2.771,Y 3.8601,Z 2,A -2.5672,B 0,C 0,E1 0.1598,E2 90.072} C_DIS
LIN {X 2.3167,Y 4.1478,Z 2,A -2.5719,B 0,C 0,E1 0.1598,E2 90.072} C_DIS
LIN {X 1.8339,Y 4.3844,Z 2,A -2.5797,B 0,C 0,E1 0.1598,E2 90.072} C_DIS
LIN {X 1.3264,Y 4.5622,Z 2,A -2.5909,B 0,C 0,E1 0.1598,E2 90.072} C_DIS
LIN {X 0.8028,Y 4.6848,Z 2,A -2.605,B 0,C 0,E1 0.1598,E2 90.072} C_DIS
LIN {X 0.2685,Y 4.7456,Z 2,A -2.6222,B 0,C 0,E1 0.1598,E2 90.072} C_DIS
LIN {X -0.2693,Y 4.7453,Z 2,A -2.642,B 0,C 0,E1 0.1598,E2 90.072} C_DIS
LIN {X -0.8038,Y 4.6854,Z 2,A -2.6643,B 0,C 0,E1 0.1598,E2 90.072} C_DIS
LIN {X -1.3277,Y 4.5639,Z 2,A -2.6887,B 0,C 0,E1 0.1598,E2 90.072} C_DIS
LIN {X -1.8347,Y 4.3843,Z 2,A -2.715,B 0,C 0,E1 0.1598,E2 90.072} C_DIS
LIN {X -2.3187,Y 4.1499,Z 2,A -2.7427,B 0,C 0,E1 0.1598,E2 90.0719} C_DIS
LIN {X -2.7726,Y 3.8613,Z 2,A -2.7715,B 0,C 0,E1 0.1598,E2 90.0719} C_DIS
LIN {X -3.1909,Y 3.5232,Z 2,A -2.8012,B 0,C 0,E1 0.1598,E2 90.0718} C_DIS
LIN {X -3.5689,Y 3.1407,Z 2,A -2.8312,B 0,C 0,E1 0.1598,E2 90.0718} C_DIS
LIN {X -3.9008,Y 2.7175,Z 2,A -2.8612,B 0,C 0,E1 0.1598,E2 90.0717} C_DIS
LIN {X -4.1816,Y 2.2588,Z 2,A -2.8909,B 0,C 0,E1 0.1598,E2 90.0717} C_DIS
LIN {X -4.4103,Y 1.772,Z 2,A -2.9198,B 0,C 0,E1 0.1598,E2 90.0716} C_DIS
LIN {X -4.5829,Y 1.2627,Z 2,A -2.9476,B 0,C 0,E1 0.1598,E2 90.0716} C_DIS
LIN {X -4.6946,Y 0.7366,Z 2,A -2.9738,B 0,C 0,E1 0.1598,E2 90.0715} C_DIS
LIN {X -4.7495,Y 0.2015,Z 2,A -2.9984,B 0,C 0,E1 0.1598,E2 90.0715} C_DIS
LIN {X -4.7399,Y -0.3362,Z 2,A -3.0206,B 0,C 0,E1 0.1598,E2 90.0715} C_DIS
LIN {X -4.6731,Y -0.8697,Z 2,A -3.0407,B 0,C 0,E1 0.1598,E2 90.0714} C_DIS
LIN {X -4.5444,Y -1.3919,Z 2,A -3.0579,B 0,C 0,E1 0.1598,E2 90.0714} C_DIS
LIN {X -4.3562,Y -1.8956,Z 2,A -3.0722,B 0,C 0,E1 0.1598,E2 90.0714} C_DIS
LIN {X -4.1154,Y -2.3764,Z 2,A -3.0837,B 0,C 0,E1 0.1598,E2 90.0714} C_DIS
LIN {X -3.82,Y -2.8256,Z 2,A -3.0918,B 0,C 0,E1 0.1598,E2 90.0714} C_DIS
LIN {X -3.4774,Y -3.2403,Z 2,A -3.0967,B 0,C 0,E1 0.1598,E2 90.0714} C_DIS
LIN {X -3.0901,Y -3.6133,Z 2,A -3.0982,B 0,C 0,E1 0.1598,E2 90.0714} C_DIS
LIN {X -2.6615,Y -3.9382,Z 2,A -3.0962,B 0,C 0,E1 0.1598,E2 90.0714} C_DIS
LIN {X -2.1994,Y -4.2134,Z 2,A -3.0908,B 0,C 0,E1 0.1598,E2 90.0714} C_DIS
LIN {X -1.7096,Y -4.4355,Z 2,A -3.0822,B 0,C 0,E1 0.1598,E2 90.0714} C_DIS
LIN {X -1.1975,Y -4.5997,Z 2,A -3.0704,B 0,C 0,E1 0.1598,E2 90.0714} C_DIS
LIN {X -0.6702,Y -4.7056,Z 2,A -3.0555,B 0,C 0,E1 0.1598,E2 90.0714} C_DIS
LIN {X 0.0001,Y -4.7539,Z 2,A -3.0329,B 0,C 0,E1 0.1598,E2 90.0715} C_DIS
Enddeposition()
LIN {X 0.0001,Y -4.7539,Z 2,A -3.0329,B 0,C 0,E1 0.1598,E2 90.0715} C_DIS
Startdeposition()
$VEL.CP = VEL_PRINT
LIN {X -0.5234,Y -5.6603,Z 2,A -3.09,B 0,C 0,E1 0.1598,E2 90.0709} C_DIS
LIN {X -1.2472,Y -5.5444,Z 2,A -3.1122,B 0,C 0,E1 0.1598,E2 90.0714} C_DIS
LIN {X -1.9509,Y -5.339,Z 2,A -3.1294,B 0,C 0,E1 0.1598,E2 90.0714} C_DIS
LIN {X -2.6224,Y -5.0444,Z 2,A -3.1416,B 0,C 0,E1 0.1598,E2 90.0714} C_DIS
LIN {X -3.2489,Y -4.6632,Z 2,A -3.1485,B 0,C 0,E1 0.1598,E2 90.0713} C_DIS
LIN {X -3.823,Y -4.2072,Z 2,A -3.1503,B 0,C 0,E1 0.1598,E2 90.0713} C_DIS
LIN {X -4.3321,Y -3.6795,Z 2,A -3.1467,B 0,C 0,E1 0.1598,E2 90.0713} C_DIS
LIN {X -4.7699,Y -3.0915,Z 2,A -3.1379,B 0,C 0,E1 0.1598,E2 90.0713} C_DIS
LIN {X -5.1275,Y -2.4515,Z 2,A -3.1241,B 0,C 0,E1 0.1598,E2 90.0712} C_DIS
LIN {X -5.4011,Y -1.7714,Z 2,A -3.1055,B 0,C 0,E1 0.1598,E2 90.0712} C_DIS
LIN {X -5.5838,Y -1.0613,Z 2,A -3.0822,B 0,C 0,E1 0.1598,E2 90.0712} C_DIS
LIN {X -5.6739,Y -0.3337,Z 2,A -3.0549,B 0,C 0,E1 0.1598,E2 90.0712} C_DIS
LIN {X -5.6393,Y 0.7603,Z 2,A -3.0073,B 0,C 0,E1 0.1598,E2 90.071} C_DIS
LIN {X -5.4512,Y 1.6179,Z 2,A -2.9645,B 0,C 0,E1 0.1598,E2 90.0713} C_DIS
LIN {X -5.0608,Y 2.6027,Z 2,A -2.9085,B 0,C 0,E1 0.1598,E2 90.0713} C_DIS
LIN {X -4.5432,Y 3.4136,Z 2,A -2.8555,B 0,C 0,E1 0.1598,E2 90.0715} C_DIS
LIN {X -4.0414,Y 3.997,Z 2,A -2.8126,B 0,C 0,E1 0.1598,E2 90.0717} C_DIS
LIN {X -3.0577,Y 4.7983,Z 2,A -2.7425,B 0,C 0,E1 0.1598,E2 90.0717} C_DIS
LIN {X -2.2838,Y 5.2074,Z 2,A -2.6969,B 0,C 0,E1 0.1598,E2 90.0719} C_DIS
LIN {X -1.499,Y 5.4838,Z 2,A -2.6564,B 0,C 0,E1 0.1598,E2 90.0719} C_DIS
LIN {X -0.6827,Y 5.6444,Z 2,A -2.6195,B 0,C 0,E1 0.1598,E2 90.0721} C_DIS
LIN {X 0.1483,Y 5.6829,Z 2,A -2.5872,B 0,C 0,E1 0.1598,E2 90.0721} C_DIS
LIN {X 0.9761,Y 5.6005,Z 2,A -2.5602,B 0,C 0,E1 0.1598,E2 90.0721} C_DIS
LIN {X 1.7825,Y 5.3964,Z 2,A -2.539,B 0,C 0,E1 0.1598,E2 90.0721} C_DIS
LIN {X 2.5513,Y 5.0791,Z 2,A -2.524,B 0,C 0,E1 0.1598,E2 90.0721} C_DIS
LIN {X 3.2646,Y 4.6513,Z 2,A -2.5157,B 0,C 0,E1 0.1598,E2 90.0721} C_DIS
LIN {X 3.9088,Y 4.1253,Z 2,A -2.5142,B 0,C 0,E1 0.1598,E2 90.0721} C_DIS
LIN {X 4.6009,Y 3.3493,Z 2,A -2.5212,B 0,C 0,E1 0.1598,E2 90.0718} C_DIS
LIN {X 4.9811,Y 2.7419,Z 2,A -2.5331,B 0,C 0,E1 0.1598,E2 90.072} C_DIS
LIN {X 5.3246,Y 1.992,Z 2,A -2.5521,B 0,C 0,E1 0.1598,E2 90.0719} C_DIS
LIN {X 5.5574,Y 1.2006,Z 2,A -2.577,B 0,C 0,E1 0.1598,E2 90.0718} C_DIS
LIN {X 5.6723,Y 0.3838,Z 2,A -2.6073,B 0,C 0,E1 0.1598,E2 90.0718} C_DIS
LIN {X 5.6683,Y -0.4412,Z 2,A -2.6424,B 0,C 0,E1 0.1598,E2 90.0717} C_DIS
LIN {X 5.5428,Y -1.2562,Z 2,A -2.6816,B 0,C 0,E1 0.1598,E2 90.0717} C_DIS
LIN {X 5.3025,Y -2.0451,Z 2,A -2.7239,B 0,C 0,E1 0.1598,E2 90.0717} C_DIS
LIN {X 4.9516,Y -2.7914,Z 2,A -2.7684,B 0,C 0,E1 0.1598,E2 90.0716} C_DIS
LIN {X 4.494,Y -3.4773,Z 2,A -2.8143,B 0,C 0,E1 0.1598,E2 90.0716} C_DIS
LIN {X 3.9453,Y -4.0931,Z 2,A -2.8606,B 0,C 0,E1 0.1598,E2 90.0716} C_DIS
LIN {X 3.3117,Y -4.6212,Z 2,A -2.9063,B 0,C 0,E1 0.1598,E2 90.0716} C_DIS
LIN {X 2.608,Y -5.0517,Z 2,A -2.9504,B 0,C 0,E1 0.1598,E2 90.0716} C_DIS
LIN {X 1.8495,Y -5.376,Z 2,A -2.992,B 0,C 0,E1 0.1598,E2 90.0716} C_DIS
LIN {X 1.0517,Y -5.5856,Z 2,A -3.0302,B 0,C 0,E1 0.1598,E2 90.0716} C_DIS
LIN {X 0.0262,Y -5.6891,Z 2,A -3.0722,B 0,C 0,E1 0.1598,E2 90.0715} C_DIS
Enddeposition()
LIN {X 0.0262,Y -5.6891,Z 2,A -3.0722,B 0,C 0,E1 0.1598,E2 90.0715} C_DIS
Startdeposition()
$VEL.CP = VEL_PRINT
LIN {X 0.5287,Y -6.5999,Z 2,A -3.0919,B 0,C 0,E1 0.1598,E2 90.0709} C_DIS
LIN {X 1.2045,Y -6.5105,Z 2,A -3.0639,B 0,C 0,E1 0.1598,E2 90.0715} C_DIS
LIN {X 1.8669,Y -6.3501,Z 2,A -3.0328,B 0,C 0,E1 0.1598,E2 90.0715} C_DIS
LIN {X 2.51,Y -6.1248,Z 2,A -2.9996,B 0,C 0,E1 0.1598,E2 90.0715} C_DIS
LIN {X 3.1276,Y -5.8362,Z 2,A -2.9647,B 0,C 0,E1 0.1598,E2 90.0715} C_DIS
LIN {X 3.7106,Y -5.4832,Z 2,A -2.9284,B 0,C 0,E1 0.1598,E2 90.0716} C_DIS
LIN {X 4.2538,Y -5.0715,Z 2,A -2.891,B 0,C 0,E1 0.1598,E2 90.0716} C_DIS
LIN {X 4.7522,Y -4.6066,Z 2,A -2.8529,B 0,C 0,E1 0.1598,E2 90.0716} C_DIS
LIN {X 5.2015,Y -4.0942,Z 2,A -2.8147,B 0,C 0,E1 0.1598,E2 90.0716} C_DIS
LIN {X 5.594,Y -3.537,Z 2,A -2.7766,B 0,C 0,E1 0.1598,E2 90.0717} C_DIS
LIN {X 5.9292,Y -2.9435,Z 2,A -2.7391,B 0,C 0,E1 0.1598,E2 90.0717} C_DIS
LIN {X 6.2022,Y -2.3189,Z 2,A -2.7026,B 0,C 0,E1 0.1598,E2 90.0717} C_DIS
LIN {X 6.4084,Y -1.6692,Z 2,A -2.6674,B 0,C 0,E1 0.1598,E2 90.0717} C_DIS
LIN {X 6.5456,Y -1.0015,Z 2,A -2.6341,B 0,C 0,E1 0.1598,E2 90.0718} C_DIS
LIN {X 6.6132,Y -0.3232,Z 2,A -2.6028,B 0,C 0,E1 0.1598,E2 90.0718} C_DIS
LIN {X 6.6097,Y 0.3583,Z 2,A -2.574,B 0,C 0,E1 0.1598,E2 90.0718} C_DIS
LIN {X 6.5391,Y 1.0363,Z 2,A -2.5479,B 0,C 0,E1 0.1598,E2 90.0719} C_DIS
LIN {X 6.3968,Y 1.7029,Z 2,A -2.5249,B 0,C 0,E1 0.1598,E2 90.0719} C_DIS
LIN {X 6.1865,Y 2.3512,Z 2,A -2.5052,B 0,C 0,E1 0.1598,E2 90.0719} C_DIS
LIN {X 5.9144,Y 2.976,Z 2,A -2.4888,B 0,C 0,E1 0.1598,E2 90.072} C_DIS
LIN {X 5.5765,Y 3.5679,Z 2,A -2.4762,B 0,C 0,E1 0.1598,E2 90.072} C_DIS
LIN {X 5.1803,Y 4.1227,Z 2,A -2.4674,B 0,C 0,E1 0.1598,E2 90.0721} C_DIS
LIN {X 4.7285,Y 4.6332,Z 2,A -2.4624,B 0,C 0,E1 0.1598,E2 90.0721} C_DIS
LIN {X 4.2261,Y 5.0939,Z 2,A -2.4615,B 0,C 0,E1 0.1598,E2 90.0721} C_DIS
LIN {X 3.6797,Y 5.5014,Z 2,A -2.4645,B 0,C 0,E1 0.1598,E2 90.0721} C_DIS
LIN {X 3.0956,Y 5.8524,Z 2,A -2.4712,B 0,C 0,E1 0.1598,E2 90.0722} C_DIS
LIN {X 2.4773,Y 6.1391,Z 2,A -2.482,B 0,C 0,E1 0.1598,E2 90.0722} C_DIS
LIN {X 1.833,Y 6.3618,Z 2,A -2.4963,B 0,C 0,E1 0.1598,E2 90.0722} C_DIS
LIN {X 1.169,Y 6.5153,Z 2,A -2.5144,B 0,C 0,E1 0.1598,E2 90.0722} C_DIS
LIN {X 0.4929,Y 6.6022,Z 2,A -2.5357,B 0,C 0,E1 0.1598,E2 90.0722} C_DIS
LIN {X -0.1885,Y 6.6159,Z 2,A -2.5603,B 0,C 0,E1 0.1598,E2 90.0722} C_DIS
LIN {X -0.868,Y 6.5626,Z 2,A -2.5876,B 0,C 0,E1 0.1598,E2 90.0722} C_DIS
LIN {X -1.5384,Y 6.4398,Z 2,A -2.6175,B 0,C 0,E1 0.1598,E2 90.0721} C_DIS
LIN {X -2.1923,Y 6.2476,Z 2,A -2.6497,B 0,C 0,E1 0.1598,E2 90.0721} C_DIS
LIN {X -2.8231,Y 5.9893,Z 2,A -2.6838,B 0,C 0,E1 0.1598,E2 90.072} C_DIS
LIN {X -3.4236,Y 5.6671,Z 2,A -2.7195,B 0,C 0,E1 0.1598,E2 90.0719} C_DIS
LIN {X -3.9871,Y 5.2836,Z 2,A -2.7564,B 0,C 0,E1 0.1598,E2 90.0719} C_DIS
LIN {X -4.5096,Y 4.8459,Z 2,A -2.7941,B 0,C 0,E1 0.1598,E2 90.0718} C_DIS
LIN {X -4.9837,Y 4.3564,Z 2,A -2.8321,B 0,C 0,E1 0.1598,E2 90.0717} C_DIS
LIN {X -5.4069,Y 3.822,Z 2,A -2.8702,B 0,C 0,E1 0.1598,E2 90.0717} C_DIS
LIN {X -5.7707,Y 3.2456,Z 2,A -2.9078,B 0,C 0,E1 0.1598,E2 90.0715} C_DIS
LIN {X -6.0747,Y 2.6355,Z 2,A -2.9447,B 0,C 0,E1 0.1598,E2 90.0715} C_DIS
LIN {X -6.3135,Y 1.997,Z 2,A -2.9803,B 0,C 0,E1 0.1598,E2 90.0714} C_DIS
LIN {X -6.4858,Y 1.3375,Z 2,A -3.0143,B 0,C 0,E1 0.1598,E2 90.0714} C_DIS
LIN {X -6.5881,Y 0.6635,Z 2,A -3.0464,B 0,C 0,E1 0.1598,E2 90.0713} C_DIS
LIN {X -6.6193,Y -0.0173,Z 2,A -3.0762,B 0,C 0,E1 0.1598,E2 90.0713} C_DIS
LIN {X -6.5844,Y -0.6981,Z 2,A -3.1036,B 0,C 0,E1 0.1598,E2 90.0713} C_DIS
LIN {X -6.4772,Y -1.3713,Z 2,A -3.128,B 0,C 0,E1 0.1598,E2 90.0712} C_DIS
LIN {X -6.301,Y -2.0298,Z 2,A -3.1492,B 0,C 0,E1 0.1598,E2 90.0712} C_DIS
LIN {X -6.059,Y -2.6669,Z 2,A -3.1671,B 0,C 0,E1 0.1598,E2 90.0712} C_DIS
LIN {X -5.7528,Y -3.2759,Z 2,A -3.1816,B 0,C 0,E1 0.1598,E2 90.0712} C_DIS
LIN {X -5.3861,Y -3.8504,Z 2,A -3.1923,B 0,C 0,E1 0.1598,E2 90.0712} C_DIS
LIN {X -4.9613,Y -4.3834,Z 2,A -3.1992,B 0,C 0,E1 0.1598,E2 90.0712} C_DIS
LIN {X -4.4842,Y -4.8704,Z 2,A -3.2022,B 0,C 0,E1 0.1598,E2 90.0712} C_DIS
LIN {X -3.96,Y -5.3061,Z 2,A -3.2014,B 0,C 0,E1 0.1598,E2 90.0712} C_DIS
LIN {X -3.3929,Y -5.6842,Z 2,A -3.1966,B 0,C 0,E1 0.1598,E2 90.0712} C_DIS
LIN {X -2.7908,Y -6.0039,Z 2,A -3.188,B 0,C 0,E1 0.1598,E2 90.0712} C_DIS
LIN {X -2.1586,Y -6.259,Z 2,A -3.1756,B 0,C 0,E1 0.1598,E2 90.0713} C_DIS
LIN {X -1.5031,Y -6.4462,Z 2,A -3.1594,B 0,C 0,E1 0.1598,E2 90.0713} C_DIS
LIN {X -0.8324,Y -6.5672,Z 2,A -3.14,B 0,C 0,E1 0.1598,E2 90.0713} C_DIS
Enddeposition()
END
